// TwinCAT 3 PLC project SlaveController
// ProgramVersion: 3.1.4024.0
// libraries:
//   Tc2_EtherCAT, * (Beckhoff Automation GmbH)
//   Tc2_Math, * (Beckhoff Automation GmbH)
//   Tc2_Standard, * (Beckhoff Automation GmbH)
//   Tc2_System, * (Beckhoff Automation GmbH)
//   Tc2_Utilities, * (Beckhoff Automation GmbH)
//   Tc3_Module, * (Beckhoff Automation GmbH)
// project tree:
//   AgiMaths/Frames/ DHTrans.TcPOU (not stored), invFrame.TcPOU (not stored), rotX.TcPOU (not stored), rotY.TcPOU (not stored), rotZ.TcPOU (not stored), transform.TcPOU (not stored)
//   AgiMaths/MatrixLib/ angAxis2Rot.TcPOU (not stored), cross.TcPOU (not stored), Det5.TcPOU (not stored), Det6.TcPOU (not stored), Det7.TcPOU (not stored), invMat2.TcPOU (not stored), invMat6.TcPOU (not stored), invMat6Old.TcPOU (not stored), invMat3.TcPOU (not stored), invMat7.TcPOU (not stored), Mat3T.TcPOU (not stored), matAdd.TcPOU (not stored), matMultiNum.TcPOU (not stored), matMultiply.TcPOU (not stored), matMultiVec.TcPOU (not stored), matSelfAdd.TcPOU (not stored), vecDot.TcPOU (not stored), vecSelfAdd.TcPOU (not stored), matSelfSub.TcPOU (not stored), matSub.TcPOU (not stored), matTranspose.TcPOU (not stored), rot2AngAxis.TcPOU (not stored), vecAdd.TcPOU (not stored), norm.TcPOU (not stored), normalize.TcPOU (not stored), vecSelfMultiNum.TcPOU (not stored), vecMultiNum.TcPOU (not stored), vecSelfSub.TcPOU (not stored), vecSub.TcPOU (not stored)
//   AgiMaths/ sign.TcPOU (not stored), addVec7.TcPOU (not stored), atan2.TcPOU (not stored), cot.TcPOU (not stored)
//   DUTs/Enum/ E_ArmLightCtrlWord.TcDUT (not stored), E_CartJointState.TcDUT, E_EndoscopeType.TcDUT (not stored), E_EndoscopePosture.TcDUT (not stored), E_InstrumentType.TcDUT (not stored), E_MasterArmState.TcDUT (not stored), E_MatchedSlaveArmIdx.TcDUT (not stored), E_SetupArmState.TcDUT (not stored), E_SlaveArmState.TcDUT (not stored), E_DriverCtrlWord.TcDUT, E_DriverOPMode.TcDUT (not stored), E_DriverStatusWord.TcDUT (not stored)
//   DUTs/Structure/MasterSlaveCommunication/ ST_MasterStatus.TcDUT (not stored), ST_SlaveStatus.TcDUT (not stored)
//   DUTs/Structure/ ST_CartInputDataPool.TcDUT (not stored), ST_EtherCATState.TcDUT (not stored), ST_InstruOnChipData.TcDUT (not stored), ST_InstruStatus.TcDUT (not stored), ST_SetupArmCtrlCmds.TcDUT (not stored), ST_SetupInputDataPool.TcDUT (not stored), ST_SlaveArmCtrlCmds.TcDUT (not stored), ST_SlaveInputDataPool.TcDUT (not stored), ST_InstruKinematicParam.TcDUT (not stored), ST_Frame.TcDUT (not stored)
//   DUTs/Structure/TasksCommunication/ ST_CartJointData.TcDUT (not stored), ST_CartMotorInput.TcDUT (not stored), ST_CartMotorOutput.TcDUT (not stored), ST_CartStatus.TcDUT (not stored), ST_CartUIData.TcDUT (not stored), ST_SetupStatus.TcDUT (not stored), ST_SetupJointData.TcDUT (not stored), ST_SlaveDynaData.TcDUT (not stored), ST_SlaveUIData.TcDUT, ST_MasterJointData.TcDUT (not stored), ST_MotorInputs.TcDUT (not stored), ST_MotorOutputs.TcDUT (not stored), ST_SlaveJointData.TcDUT (not stored), ST_SafetyData.TcDUT (not stored)
//   DUTs/Structure/UICommunication/ ST_cartOperation.TcDUT (not stored), ST_instruInfomation.TcDUT (not stored), ST_robotStateMachine.TcDUT (not stored), ST_uiControl.TcDUT (not stored)
//   DUTs/Type/ Mat23.TcDUT (not stored), Mat2d.TcDUT (not stored), Mat32.TcDUT (not stored), Mat34.TcDUT (not stored), Mat53.TcDUT (not stored), Mat37.TcDUT (not stored), Mat43.TcDUT (not stored), Mat45.TcDUT (not stored), Mat35.TcDUT (not stored), Mat4d.TcDUT (not stored), Mat5d.TcDUT (not stored), Mat67.TcDUT (not stored), Mat6d.TcDUT (not stored), Mat76.TcDUT (not stored), Mat7d.TcDUT (not stored), Vec13d.TcDUT (not stored), Vec13di.TcDUT (not stored), Vec2d.TcDUT (not stored), Vec2i.TcDUT (not stored), Vec4b.TcDUT (not stored), Vec4d.TcDUT (not stored), Vec4i.TcDUT (not stored), Vec5b.TcDUT (not stored), Vec5d.TcDUT (not stored), Vec5i.TcDUT (not stored), Vec6b.TcDUT (not stored), Vec6i.TcDUT (not stored), Vec8b.TcDUT (not stored), Vec8d.TcDUT (not stored), Vec8di.TcDUT (not stored), Vec8i.TcDUT (not stored), Mat3d.TcDUT (not stored), Vec3d.TcDUT (not stored), Vec6d.TcDUT (not stored), Vec7d.TcDUT (not stored), Vec7i.TcDUT (not stored)
//   FBs_Auxiliary/ FB_cartJntDisenableDetect.TcPOU (not stored), FB_cartJntEnableDetect.TcPOU (not stored), FB_InstruNearDetect.TcPOU (not stored), FB_IOCheck.TcPOU (not stored), FB_IOToggleCheck.TcPOU (not stored), FB_rotaButtonDetect.TcPOU (not stored), FB_setupAdjustDetect.TcPOU (not stored), FB_setupJnt5AdjustDetect.TcPOU, FB_masterConnectionCheck.TcPOU (not stored), FB_TON.TcPOU (not stored), FB_trocarDetect.TcPOU (not stored), FB_PanelDetect.TcPOU, FB_InstrumentDetect.TcPOU, FB_AdjustDetect.TcPOU (not stored)
//   FBs_BasicControllers/ FB_dither.TcPOU (not stored), FB_BasicInstruControl.TcPOU (not stored), FBMacroJntControl.TcPOU (not stored), FB_UltrosonicKnifeControl.TcPOU (not stored), FB_PID.TcPOU (not stored)
//   FBs_CartControlles/ FB_CartCtrlAdjust.TcPOU, FB_CartCtrlAsepticDeploy.TcPOU (not stored), FB_CartCtrlBase.TcPOU (not stored), FB_CartCtrlError.TcPOU (not stored), FB_CartCtrlInit.TcPOU (not stored), FB_CartCtrlInSurgery.TcPOU (not stored), FB_CartCtrlMotionCar.TcPOU (not stored), FB_CartCtrlReady.TcPOU (not stored), FB_CartCtrlRotaOverhang.TcPOU (not stored), FB_CartCtrlSlowDown.TcPOU, FB_CartCtrlStandColuAdjust.TcPOU (not stored), FB_CartSupporLeg.TcPOU, I_CartJointCtrl.TcIO (not stored)
//   FBs_RobotDynamics/ FB_SlaveDynamic.TcPOU (not stored), FB_SlaveGravity.TcPOU (not stored), FB_SetupGravity.TcPOU
//   FBs_Robots/ FB_CartJoint.TcPOU, FB_CartRobot.TcPOU, FB_Instrument.TcPOU, FB_JointBase.TcPOU, FB_SetupArm.TcPOU, FB_SlaveCart.TcPOU, FB_SlaveJoint.TcPOU, FB_SetupJoint.TcPOU (not stored), FB_SetupRobot.TcPOU (not stored), FB_SlaveArm.TcPOU (not stored), FB_SlaveRobot.TcPOU
//   FBs_SetupControllers/ FB_SetupCtrlDisable.TcPOU (not stored), FB_SetupCtrlJnt5GraCali.TcPOU (not stored), FB_SetupCtrlHold.TcPOU (not stored), FB_SetupCtrlManualAdjust.TcPOU, FB_SetupCtrlPerformance.TcPOU (not stored), FB_SetupArmCtrlBase.TcPOU (not stored), FB_SetupCtrlAutoAdjust.TcPOU (not stored), FB_SetupCtrlCart.TcPOU (not stored), FB_SetupCtrlError.TcPOU (not stored), FB_SetupCtrlJnt3GraCali.TcPOU (not stored), FB_SetupCtrlInit.TcPOU (not stored), FB_SetupCtrlPackage.TcPOU (not stored), FB_SetupCtrlSelfCheck.TcPOU (not stored), I_SetupArmCtrl.TcIO (not stored)
//   FBs_SlaveControllers/ FB_SlaveCtrlDisable.TcPOU (not stored), FB_SlaveCtrlInstruInvasion.TcPOU (not stored), FB_SlaveCtrlInstruRetract.TcPOU (not stored), FB_SlaveCtrlInstruCali.TcPOU (not stored), FB_SlaveCtrlPerformance.TcPOU (not stored), FB_SlaveCtrlScopeToggle.TcPOU (not stored), FB_SlaveCtrlStop.TcPOU (not stored), FB_SlaveCtrlTest.TcPOU (not stored), FB_SlaveCtrlPackage.TcPOU (not stored), FB_SlaveCtrlEndoscope.TcPOU (not stored), FB_SlaveCtrlCart.TcPOU (not stored), FB_SlaveCtrlScopeReady.TcPOU (not stored), FB_SlaveCtrlSelfCheck.TcPOU, FB_SlaveCtrlError.TcPOU (not stored), FB_SlaveCtrlInstruReady.TcPOU (not stored), FB_SlaveCtrlMasterSlave.TcPOU, FB_SlaveCtrlMountInstru.TcPOU, FB_SlaveCtrlAdjust.TcPOU (not stored), FB_SlaveCtrlMountPanel.TcPOU (not stored), FB_SlaveCtrlPanelReady.TcPOU (not stored), FB_SlaveCtrlGraCali.TcPOU (not stored), FB_SlaveCtrlInit.TcPOU (not stored), FB_SlaveCtrlStandBy.TcPOU (not stored), FB_SlaveArmCtrlBase.TcPOU (not stored), I_SlaveArmCtrl.TcIO (not stored)
//   FBs_TrajectoryPlanning/ FB_BasicDoubleS.TcPOU (not stored), FB_trajBase.TcPOU (not stored), FB_TrajMoveJ.TcPOU (not stored), FB_setupTrajMoveJ.TcPOU (not stored), linear_trajectory_with_quintic_polynomial_blends.TcPOU (not stored), quintic_spline_curve.TcPOU (not stored), Quintic_spline_curve_factor.TcPOU (not stored), TrapezoIDal_velocity_trajectory.TcPOU (not stored)
//   FBs_TrajectoryPlanning/OTG/ FB_secOrdTrajFilter.TcPOU (not stored), FB_thirdOrdTrajFilter.TcPOU (not stored)
//   FBs_Filters/ FB_LowPassFilter.TcPOU (not stored)
//   GVLs/CartJoints/ GVL_CartControlParameters.TcGVL, GVL_CartJointEncoderCaliData.TcGVL, GVL_CartMotorParameters.TcGVL
//   GVLs/configs/robot3/ GVL_CartJointEncoderCaliData_3.TcGVL (not stored), GVL_SetupArmDynamics_3.TcGVL (not stored), GVL_SlaveArmDynamics_3.TcGVL (not stored), GVL_SetupJointEncoderCaliData_3.TcGVL (not stored), GVL_SlaveJointEncoderCaliData_3.TcGVL (not stored)
//   GVLs/configs/robot5/ GVL_CartJointEncoderCaliData_5.TcGVL (not stored), GVL_SetupArmDynamics_5.TcGVL (not stored), GVL_SlaveArmDynamics_5.TcGVL (not stored), GVL_SetupJointEncoderCaliData_5.TcGVL (not stored), GVL_SlaveJointEncoderCaliData_5.TcGVL (not stored)
//   GVLs/configs/robot4/ GVL_SetupArmDynamics_4.TcGVL (not stored), GVL_SetupJointEncoderCaliData_4.TcGVL (not stored), GVL_SlaveArmDynamics_4.TcGVL (not stored), GVL_SlaveJointEncoderCaliData_4.TcGVL (not stored)
//   GVLs/configs/robot6/ GVL_CartJointEncoderCaliData_6.TcGVL (not stored), GVL_SetupArmDynamics_6.TcGVL (not stored), GVL_SetupJointEncoderCaliData_6.TcGVL (not stored), GVL_SlaveArmDynamics_6.TcGVL (not stored), GVL_SlaveJointEncoderCaliData_6.TcGVL (not stored)
//   GVLs/ GVL_InstruCtrlParams.TcGVL, GVL_interactUI.TcGVL, GVL_MathDefine.TcGVL (not stored), GVL_SafetyLogData.TcGVL, GVL_SafetyParameters.TcGVL, GVL_SystemParameters.TcGVL
//   GVLs/SetupArms/ GVL_SetupArmDynamics.TcGVL (not stored), GVL_SetupJointEncoderCaliData.TcGVL, GVL_SetupMotorParameters.TcGVL, GVL_SetupArmKinematic.TcGVL (not stored), GVL_SetupControlParameters.TcGVL (not stored)
//   GVLs/SlaveArms/ GVL_SlaveArmDynamics.TcGVL (not stored), GVL_SlaveArmKinematic.TcGVL (not stored), GVL_SlaveControlParameters.TcGVL, GVL_SlaveJointEncoderCaliData.TcGVL, GVL_SlaveMotorParameters.TcGVL
//   Mains/ CartControl.TcPOU, SafetyCheck.TcPOU, SetupArmControl.TcPOU (not stored), SlaveArmControl.TcPOU, RobotDynamics.TcPOU (not stored)
//   SafetyCheck/ ASSERT.TcPOU (not stored), Fb_dataRecord.TcPOU (not stored), FB_EtherCATCheck.TcPOU (not stored), Fb_SafetyCheck.TcPOU, FB_Writer.TcPOU (not stored)
//   SafetyCheck/ErrRecord/ checkDelay.TcDUT (not stored), checkDelayTime.TcDUT, checkInputVariable.TcDUT (not stored), checkPermit.TcDUT (not stored), ST_Buffer.TcDUT (not stored), T_Buffer.TcDUT (not stored)
//   Sandbox/ FB_SlaveCtrlMasterSlave_bak1.TcPOU (not stored), FB_SlaveCtrlMasterSlave_bak2.TcPOU (not stored)
//   / TaskCartControl.TcTTO (not stored), TaskDynamic.TcTTO (not stored), TaskSafetyCheck.TcTTO (not stored), TaskSetupArmControl.TcTTO (not stored), TaskSlaveArmControl.TcTTO (not stored)
// real-time tasks:
//   TASK TaskSlaveArmControl: cycle T#250us, priority 1, ADS port 350
//   TASK TaskDynamic: cycle T#1ms, priority 2, ADS port 351
//   TASK TaskSetupArmControl: cycle T#1ms, priority 3, ADS port 352
//   TASK TaskSafetyCheck: cycle T#1ms, priority 6, ADS port 353
//   TASK TaskCartControl: cycle T#1ms, priority 4, ADS port 354
// I/O:
//   DEVICE CU2508
//   DEVICE Cart, AmsNetId 169.254.45.61.8.1
//     CartJoint5 [MDDLN55BE]
//     CartJoint3 [MDDLN55BE]
//     CartJoint4 [MDDLN55BE]
//     CartJoint1 [AX58200_MotorControl_for_1axis]
//     CartJoint2 [AX58200_MotorControl_for_1axis]
//     RS232 [AX58200_CANFD]
//     CartJoint6 [AX58200_MotorControl_for_1axis]
//     CartJoint7 [AX58200_MotorControl_for_1axis]
//     CartJoint8 [AX58200_MotorControl_for_1axis]
//   DEVICE MSCommunication, AmsNetId 169.254.186.39.3.1
//     Term 20 (EK1100) [EK1100 EtherCAT Coupler (2A E-Bus)]
//       Term 21 (EL6695) [EL6695 EtherCAT Bridge terminal (Primary)]
//       Term 8 (EL9011) [EL9011 End Terminal]
//     Term 22 (EK1100) [EK1100 EtherCAT Coupler (2A E-Bus)]
//       Term 23 (EL6070) [EL6070 1Ch. Licensing-Terminal]
//       Term 24 (EL1008) [EL1008 8Ch. Dig. Input 24V, 3ms]
//       Term 25 (EL2008) [EL2008 8Ch. Dig. Output 24V, 0.5A]
//       Term 26 (EL3004) [EL3004 4Ch. Ana. Input +/-10V] (disabled)
//       Term 9 (EL9011) [EL9011 End Terminal]
//   DEVICE SlaveArm1, AmsNetId 169.254.223.120.10.1
//     Box 25 (CU2508) [CU2508 Ethernet Port]
//     SetupJoint12 [AX58200_MotorControl_for_1axis]
//     SetupJoint3 [AX58200_MotorControl_for_1axis]
//     SetupJoint45 [AX58200_MotorControl_Slave45]
//     SlaveJoint1 [AX58200_MotorControl_for_1axis]
//     SlaveJoint2 [AX58200_MotorControl_for_1axis]
//     SlaveJoint3 [AX58200_MotorControl_for_1axis]
//     SlaveJoint45 [AX58200_MotorControl_3axis]
//     SlaveJoint678 [AX58200_MotorControl_3axis]
//   DEVICE SlaveArm2, AmsNetId 192.168.2.91.4.1
//     Box 25 (CU2508) [CU2508 Ethernet Port]
//     SetupJoint12 [AX58200_MotorControl_for_1axis]
//     SetupJoint3 [AX58200_MotorControl_for_1axis]
//     SetupJoint45 [AX58200_MotorControl_Slave45]
//     SlaveJoint1 [AX58200_MotorControl_for_1axis]
//     SlaveJoint2 [AX58200_MotorControl_for_1axis]
//     SlaveJoint3 [AX58200_MotorControl_for_1axis]
//     SlaveJoint45 [AX58200_MotorControl_3axis]
//     SlaveJoint678 [AX58200_MotorControl_3axis]
//   DEVICE SlaveArm3, AmsNetId 192.168.2.91.6.1
//     Box 17 (CU2508) [CU2508 Ethernet Port]
//     SetupJoint12 [AX58200_MotorControl_for_1axis]
//     SetupJoint3 [AX58200_MotorControl_for_1axis]
//     SetupJoint45 [AX58200_MotorControl_Slave45]
//     SlaveJoint1 [AX58200_MotorControl_for_1axis]
//     SlaveJoint2 [AX58200_MotorControl_for_1axis]
//     SlaveJoint3 [AX58200_MotorControl_for_1axis]
//     SlaveJoint45 [AX58200_MotorControl_3axis]
//     SlaveJoint678 [AX58200_MotorControl_3axis]
//   DEVICE SlaveArm4, AmsNetId 192.168.2.91.5.1
//     Box 9 (CU2508) [CU2508 Ethernet Port]
//     SetupJoint12 [AX58200_MotorControl_for_1axis]
//     SetupJoint3 [AX58200_MotorControl_for_1axis]
//     SetupJoint45 [AX58200_MotorControl_Slave45]
//     SlaveJoint1 [AX58200_MotorControl_for_1axis]
//     SlaveJoint2 [AX58200_MotorControl_for_1axis]
//     SlaveJoint3 [AX58200_MotorControl_for_1axis]
//     SlaveJoint45 [AX58200_MotorControl_3axis]
//     SlaveJoint678 [AX58200_MotorControl_3axis]
// variable links:
//   SlaveController/SlaveController Instance <-> Cart/CartJoint1
//     TaskCartControl Inputs/CartControl.m_cartRobot.m_slaveCart.m_cartJoints[1].m_motorInputs/m_current <-> TxPdoMappingCspCsv/Torque actual value
//     TaskCartControl Inputs/CartControl.m_cartRobot.m_slaveCart.m_cartJoints[1].m_motorInputs/m_motorEncoder <-> TxPdoMappingCspCsv/Position actual value
//     TaskCartControl Inputs/CartControl.m_cartRobot.m_slaveCart.m_cartJoints[1].m_motorInputs/m_statusWord <-> TxPdoMappingCspCsv/Statusword
//     TaskCartControl Inputs/CartControl.m_cartRobot.m_slaveCart.m_cartJoints[5].m_motorInputs/m_linkEncoder <-> TxPdoMappingCspCsv/ENC2
//     TaskCartControl Outputs/CartControl.m_cartRobot.m_slaveCart.m_cartJoints[1].m_motorOutputs/m_cmdCurrent <-> RxPdoMappingCspCsv/Target torque
//     TaskCartControl Outputs/CartControl.m_cartRobot.m_slaveCart.m_cartJoints[1].m_motorOutputs/m_cmdMotorEncoder <-> RxPdoMappingCspCsv/Target position
//     TaskCartControl Outputs/CartControl.m_cartRobot.m_slaveCart.m_cartJoints[1].m_motorOutputs/m_controlWord <-> RxPdoMappingCspCsv/Controlword
//     TaskCartControl Outputs/CartControl.m_cartRobot.m_slaveCart.m_cartJoints[1].m_motorOutputs/m_opMode <-> RxPdoMappingCspCsv/Modes of operation
//   SlaveController/SlaveController Instance <-> Cart/CartJoint2
//     TaskCartControl Inputs/CartControl.m_cartRobot.m_slaveCart.m_cartJoints[2].m_motorInputs/m_current <-> TxPdoMappingCspCsv/Torque actual value
//     TaskCartControl Inputs/CartControl.m_cartRobot.m_slaveCart.m_cartJoints[2].m_motorInputs/m_motorEncoder <-> TxPdoMappingCspCsv/Position actual value
//     TaskCartControl Inputs/CartControl.m_cartRobot.m_slaveCart.m_cartJoints[2].m_motorInputs/m_statusWord <-> TxPdoMappingCspCsv/Statusword
//     TaskCartControl Outputs/CartControl.m_cartRobot.m_slaveCart.m_cartJoints[2].m_motorOutputs/m_cmdCurrent <-> RxPdoMappingCspCsv/Target torque
//     TaskCartControl Outputs/CartControl.m_cartRobot.m_slaveCart.m_cartJoints[2].m_motorOutputs/m_cmdMotorEncoder <-> RxPdoMappingCspCsv/Target position
//     TaskCartControl Outputs/CartControl.m_cartRobot.m_slaveCart.m_cartJoints[2].m_motorOutputs/m_controlWord <-> RxPdoMappingCspCsv/Controlword
//     TaskCartControl Outputs/CartControl.m_cartRobot.m_slaveCart.m_cartJoints[2].m_motorOutputs/m_opMode <-> RxPdoMappingCspCsv/Modes of operation
//   SlaveController/SlaveController Instance <-> Cart/CartJoint3
//     TaskCartControl Inputs/CartControl.m_cartRobot.m_slaveCart.m_cartJoints[3].m_cartMotorVelSongxia <-> Transmit PDO mapping 2/Velocity actual value
//     TaskCartControl Inputs/CartControl.m_cartRobot.m_slaveCart.m_cartJoints[3].m_motorInputs/m_statusWord <-> Transmit PDO mapping 2/Statusword
//     TaskCartControl Outputs/CartControl.m_cartRobot.m_slaveCart.m_cartJoints[3].m_cartMotorOutput/m_cmdVelMax <-> Receive PDO mapping 2/Max motor speed
//     TaskCartControl Outputs/CartControl.m_cartRobot.m_slaveCart.m_cartJoints[3].m_cartMotorOutput/m_cmdVelMzVelMode <-> Receive PDO mapping 2/Target velocity
//     TaskCartControl Outputs/CartControl.m_cartRobot.m_slaveCart.m_cartJoints[3].m_motorOutputs/m_controlWord <-> Receive PDO mapping 2/Controlword
//     TaskCartControl Outputs/CartControl.m_cartRobot.m_slaveCart.m_cartJoints[3].m_motorOutputs/m_opMode <-> Receive PDO mapping 2/Modes of operation
//   SlaveController/SlaveController Instance <-> Cart/CartJoint4
//     TaskCartControl Inputs/CartControl.m_cartRobot.m_slaveCart.m_cartJoints[4].m_cartMotorVelSongxia <-> Transmit PDO mapping 2/Velocity actual value
//     TaskCartControl Inputs/CartControl.m_cartRobot.m_slaveCart.m_cartJoints[4].m_motorInputs/m_statusWord <-> Transmit PDO mapping 2/Statusword
//     TaskCartControl Outputs/CartControl.m_cartRobot.m_slaveCart.m_cartJoints[4].m_cartMotorOutput/m_cmdVelMax <-> Receive PDO mapping 2/Max motor speed
//     TaskCartControl Outputs/CartControl.m_cartRobot.m_slaveCart.m_cartJoints[4].m_cartMotorOutput/m_cmdVelMzVelMode <-> Receive PDO mapping 2/Target velocity
//     TaskCartControl Outputs/CartControl.m_cartRobot.m_slaveCart.m_cartJoints[4].m_motorOutputs/m_controlWord <-> Receive PDO mapping 2/Controlword
//     TaskCartControl Outputs/CartControl.m_cartRobot.m_slaveCart.m_cartJoints[4].m_motorOutputs/m_opMode <-> Receive PDO mapping 2/Modes of operation
//   SlaveController/SlaveController Instance <-> Cart/CartJoint5
//     TaskCartControl Inputs/CartControl.m_cartRobot.m_slaveCart.m_cartJoints[5].m_motorInputs/m_motorEncoder <-> Transmit PDO mapping 1/Position actual value
//     TaskCartControl Inputs/CartControl.m_cartRobot.m_slaveCart.m_cartJoints[5].m_motorInputs/m_statusWord <-> Transmit PDO mapping 1/Statusword
//     TaskCartControl Outputs/CartControl.m_cartRobot.m_slaveCart.m_cartJoints[5].m_motorOutputs/m_cmdMotorEncoder <-> Receive PDO mapping 1/Target position
//     TaskCartControl Outputs/CartControl.m_cartRobot.m_slaveCart.m_cartJoints[5].m_motorOutputs/m_controlWord <-> Receive PDO mapping 1/Controlword
//     TaskCartControl Outputs/CartControl.m_cartRobot.m_slaveCart.m_cartJoints[5].m_motorOutputs/m_opMode <-> Receive PDO mapping 1/Modes of operation
//   SlaveController/SlaveController Instance <-> Cart/CartJoint6
//     TaskCartControl Inputs/CartControl.m_cartRobot.m_slaveCart.m_cartJoints[6].m_motorInputs/m_current <-> TxPdoMappingCspCsv/Torque actual value
//     TaskCartControl Inputs/CartControl.m_cartRobot.m_slaveCart.m_cartJoints[6].m_motorInputs/m_linkEncoder <-> TxPdoMappingCspCsv/ENC2
//     TaskCartControl Inputs/CartControl.m_cartRobot.m_slaveCart.m_cartJoints[6].m_motorInputs/m_motorEncoder <-> TxPdoMappingCspCsv/Position actual value
//     TaskCartControl Inputs/CartControl.m_cartRobot.m_slaveCart.m_cartJoints[6].m_motorInputs/m_statusWord <-> TxPdoMappingCspCsv/Statusword
//     TaskCartControl Outputs/CartControl.m_cartRobot.m_openHorizonLaser <-> RxPdoMappingCspCsv/Target velocity
//     TaskCartControl Outputs/CartControl.m_cartRobot.m_slaveCart.m_cartJoints[6].m_motorOutputs/m_cmdCurrent <-> RxPdoMappingCspCsv/Target torque
//     TaskCartControl Outputs/CartControl.m_cartRobot.m_slaveCart.m_cartJoints[6].m_motorOutputs/m_cmdMotorEncoder <-> RxPdoMappingCspCsv/Target position
//     TaskCartControl Outputs/CartControl.m_cartRobot.m_slaveCart.m_cartJoints[6].m_motorOutputs/m_controlWord <-> RxPdoMappingCspCsv/Controlword
//     TaskCartControl Outputs/CartControl.m_cartRobot.m_slaveCart.m_cartJoints[6].m_motorOutputs/m_opMode <-> RxPdoMappingCspCsv/Modes of operation
//   SlaveController/SlaveController Instance <-> Cart/CartJoint7
//     TaskCartControl Inputs/CartControl.m_cartRobot.m_slaveCart.m_cartJoints[7].m_motorInputs/m_current <-> TxPdoMappingCspCsv/Torque actual value
//     TaskCartControl Inputs/CartControl.m_cartRobot.m_slaveCart.m_cartJoints[7].m_motorInputs/m_driverError <-> TxPdoMappingCspCsv/digital input
//     TaskCartControl Inputs/CartControl.m_cartRobot.m_slaveCart.m_cartJoints[7].m_motorInputs/m_linkEncoder <-> TxPdoMappingCspCsv/ENC2
//     TaskCartControl Inputs/CartControl.m_cartRobot.m_slaveCart.m_cartJoints[7].m_motorInputs/m_motorEncoder <-> TxPdoMappingCspCsv/Position actual value
//     TaskCartControl Inputs/CartControl.m_cartRobot.m_slaveCart.m_cartJoints[7].m_motorInputs/m_statusWord <-> TxPdoMappingCspCsv/Statusword
//     TaskCartControl Outputs/CartControl.m_cartRobot.m_slaveCart.m_cartJoints[7].m_motorOutputs/m_cmdCurrent <-> RxPdoMappingCspCsv/Target torque
//     TaskCartControl Outputs/CartControl.m_cartRobot.m_slaveCart.m_cartJoints[7].m_motorOutputs/m_cmdMotorEncoder <-> RxPdoMappingCspCsv/Target position
//     TaskCartControl Outputs/CartControl.m_cartRobot.m_slaveCart.m_cartJoints[7].m_motorOutputs/m_controlWord <-> RxPdoMappingCspCsv/Controlword
//     TaskCartControl Outputs/CartControl.m_cartRobot.m_slaveCart.m_cartJoints[7].m_motorOutputs/m_opMode <-> RxPdoMappingCspCsv/Modes of operation
//   SlaveController/SlaveController Instance <-> Cart/CartJoint8
//     TaskCartControl Inputs/CartControl.m_cartRobot.m_slaveCart.m_cartJoints[8].m_motorInputs/m_current <-> TxPdoMappingCspCsv/Torque actual value
//     TaskCartControl Inputs/CartControl.m_cartRobot.m_slaveCart.m_cartJoints[8].m_motorInputs/m_driverError <-> TxPdoMappingCspCsv/digital input
//     TaskCartControl Inputs/CartControl.m_cartRobot.m_slaveCart.m_cartJoints[8].m_motorInputs/m_linkEncoder <-> TxPdoMappingCspCsv/ENC2
//     TaskCartControl Inputs/CartControl.m_cartRobot.m_slaveCart.m_cartJoints[8].m_motorInputs/m_motorEncoder <-> TxPdoMappingCspCsv/Position actual value
//     TaskCartControl Inputs/CartControl.m_cartRobot.m_slaveCart.m_cartJoints[8].m_motorInputs/m_statusWord <-> TxPdoMappingCspCsv/Statusword
//     TaskCartControl Outputs/CartControl.m_cartRobot.m_openCrossLaser <-> RxPdoMappingCspCsv/Target velocity
//     TaskCartControl Outputs/CartControl.m_cartRobot.m_slaveCart.m_cartJoints[8].m_motorOutputs/m_cmdCurrent <-> RxPdoMappingCspCsv/Target torque
//     TaskCartControl Outputs/CartControl.m_cartRobot.m_slaveCart.m_cartJoints[8].m_motorOutputs/m_cmdMotorEncoder <-> RxPdoMappingCspCsv/Target position
//     TaskCartControl Outputs/CartControl.m_cartRobot.m_slaveCart.m_cartJoints[8].m_motorOutputs/m_controlWord <-> RxPdoMappingCspCsv/Controlword
//     TaskCartControl Outputs/CartControl.m_cartRobot.m_slaveCart.m_cartJoints[8].m_motorOutputs/m_opMode <-> RxPdoMappingCspCsv/Modes of operation
//   SlaveController/SlaveController Instance <-> Cart/RS232
//     TaskCartControl Inputs/CartControl.m_cartRobot.m_slaveCart.m_driveForce[1] <-> TxPdoMappingCspCsv/FX
//     TaskCartControl Inputs/CartControl.m_cartRobot.m_slaveCart.m_driveForce[2] <-> TxPdoMappingCspCsv/FY
//     TaskCartControl Inputs/CartControl.m_cartRobot.m_slaveCart.m_driveForce[3] <-> TxPdoMappingCspCsv/MZ
//     TaskCartControl Inputs/CartControl.m_cartRobot.m_slaveCart.m_joystickSignalIO[1] <-> TxPdoMappingCspCsv/D
//     TaskCartControl Inputs/CartControl.m_cartRobot.m_slaveCart.m_joystickSignalIO[2] <-> TxPdoMappingCspCsv/B
//     TaskCartControl Inputs/CartControl.m_cartRobot.m_slaveCart.m_joystickSignalIO[3] <-> TxPdoMappingCspCsv/A
//     TaskCartControl Inputs/CartControl.m_cartRobot.m_slaveCart.m_joystickSignalIO[4] <-> TxPdoMappingCspCsv/C
//   SlaveController/SlaveController Instance <-> MSCommunication/Term 20 (EK1100)/Term 21 (EL6695)
//     TaskSafetyCheck Inputs/SafetyCheck.m_masterRobotData <-> IO Inputs/MasterRobotData
//     TaskSlaveArmControl Inputs/SlaveArmControl.m_masterRobotData <-> IO Inputs/MasterRobotData
//     TaskSlaveArmControl Outputs/SlaveArmControl.m_slaveRobotData <-> IO Outputs/SlaveRobotData
//   SlaveController/SlaveController Instance <-> MSCommunication/Term 22 (EK1100)/Term 24 (EL1008)
//     TaskCartControl Inputs/CartControl.m_cartRobot.m_carHandChassisDriveUnlock[1] <-> Channel 5/Input
//     TaskCartControl Inputs/CartControl.m_cartRobot.m_carHandChassisDriveUnlock[2] <-> Channel 6/Input
//     TaskCartControl Inputs/CartControl.m_cartRobot.m_slaveCart.m_drivingLeverSensorAuto <-> Channel 8/Input
//     TaskCartControl Inputs/CartControl.m_cartRobot.m_slaveCart.m_drivingLeverSensorManual <-> Channel 7/Input
//     TaskCartControl Inputs/CartControl.m_cartRobot.m_slaveCart.m_stabilizFootSensorLeft <-> Channel 3/Input
//     TaskCartControl Inputs/CartControl.m_cartRobot.m_slaveCart.m_stabilizFootSensorRight <-> Channel 4/Input
//     TaskSafetyCheck Inputs/SafetyCheck.m_emergencyStopButton <-> Channel 2/Input
//     TaskSlaveArmControl Inputs/SafetyCheck.m_stopButton <-> Channel 1/Input
//   SlaveController/SlaveController Instance <-> MSCommunication/Term 22 (EK1100)/Term 25 (EL2008)
//     TaskCartControl Outputs/CartControl.m_cartRobot.m_slaveCart.m_screwBreak <-> Channel 5/Output
//     TaskSafetyCheck Outputs/SafetyCheck.m_warningTone[{1..4}] <-> Channel {1..4}/Output  (4 links)
//   SlaveController/SlaveController Instance <-> SlaveArm1/SetupJoint12
//     TaskSetupArmControl Inputs/SetupArmControl.m_setupRobot.m_setupArms[1].m_joints[1].m_motorInputs/m_linkEncoder <-> TxPdoMappingCspCsv/ENC2
//     TaskSetupArmControl Inputs/SetupArmControl.m_setupRobot.m_setupArms[1].m_joints[1].m_motorInputs/m_statusWord <-> TxPdoMappingCspCsv/Statusword
//     TaskSetupArmControl Inputs/SetupArmControl.m_setupRobot.m_setupArms[1].m_joints[2].m_motorInputs/m_statusWord <-> TxPdoMappingCspCsv/Statusword
//     TaskSetupArmControl Inputs/SetupArmControl.m_setupRobot.m_setupArms[1].m_joints[2].m_motorInputs/m_linkEncoder <-> TxPdoMappingCspCsv/Velocity actual value
//     TaskSetupArmControl Outputs/SetupArmControl.m_setupRobot.m_setupArms[1].m_joints[1].m_motorOutputs/m_controlWord <-> RxPdoMappingCspCsv/Controlword
//     TaskSetupArmControl Outputs/SetupArmControl.m_setupRobot.m_setupArms[1].m_joints[1].m_motorOutputs/m_opMode <-> RxPdoMappingCspCsv/Modes of operation
//   SlaveController/SlaveController Instance <-> SlaveArm1/SetupJoint3
//     TaskSetupArmControl Inputs/SetupArmControl.m_setupRobot.m_setupArms[1].m_joints[3].m_motorInputs/m_current <-> TxPdoMappingCspCsv/Torque actual value
//     TaskSetupArmControl Inputs/SetupArmControl.m_setupRobot.m_setupArms[1].m_joints[3].m_motorInputs/m_linkEncoder <-> TxPdoMappingCspCsv/ENC2
//     TaskSetupArmControl Inputs/SetupArmControl.m_setupRobot.m_setupArms[1].m_joints[3].m_motorInputs/m_motorEncoder <-> TxPdoMappingCspCsv/Position actual value
//     TaskSetupArmControl Inputs/SetupArmControl.m_setupRobot.m_setupArms[1].m_joints[3].m_motorInputs/m_statusWord <-> TxPdoMappingCspCsv/Statusword
//     TaskSetupArmControl Outputs/SetupArmControl.m_setupRobot.m_setupArms[1].m_joints[3].m_motorOutputs/m_cmdCurrent <-> RxPdoMappingCspCsv/Target torque
//     TaskSetupArmControl Outputs/SetupArmControl.m_setupRobot.m_setupArms[1].m_joints[3].m_motorOutputs/m_cmdMotorEncoder <-> RxPdoMappingCspCsv/Target position
//     TaskSetupArmControl Outputs/SetupArmControl.m_setupRobot.m_setupArms[1].m_joints[3].m_motorOutputs/m_controlWord <-> RxPdoMappingCspCsv/Controlword
//     TaskSetupArmControl Outputs/SetupArmControl.m_setupRobot.m_setupArms[1].m_joints[3].m_motorOutputs/m_opMode <-> RxPdoMappingCspCsv/Modes of operation
//   SlaveController/SlaveController Instance <-> SlaveArm1/SetupJoint45
//     TaskSetupArmControl Inputs/SetupArmControl.m_setupRobot.m_setupArms[1].m_joints[4].m_motorInputs/m_current <-> TxPdoMappingCspCsv/Torque actual value
//     TaskSetupArmControl Inputs/SetupArmControl.m_setupRobot.m_setupArms[1].m_joints[4].m_motorInputs/m_linkEncoder <-> TxPdoMappingCspCsv/ENC2
//     TaskSetupArmControl Inputs/SetupArmControl.m_setupRobot.m_setupArms[1].m_joints[4].m_motorInputs/m_motorEncoder <-> TxPdoMappingCspCsv/Position actual value
//     TaskSetupArmControl Inputs/SetupArmControl.m_setupRobot.m_setupArms[1].m_joints[4].m_motorInputs/m_statusWord <-> TxPdoMappingCspCsv/Statusword
//     TaskSetupArmControl Inputs/SetupArmControl.m_setupRobot.m_setupArms[1].m_joints[5].m_motorInputs/m_current <-> TxPdoMappingCspCsv/Torque actual value for aix2
//     TaskSetupArmControl Inputs/SetupArmControl.m_setupRobot.m_setupArms[1].m_joints[5].m_motorInputs/m_linkEncoder <-> TxPdoMappingCspCsv/ENC2 for aix2
//     TaskSetupArmControl Inputs/SetupArmControl.m_setupRobot.m_setupArms[1].m_joints[5].m_motorInputs/m_motorEncoder <-> TxPdoMappingCspCsv/Position actual value for aix2
//     TaskSetupArmControl Inputs/SetupArmControl.m_setupRobot.m_setupArms[1].m_joints[5].m_motorInputs/m_statusWord <-> TxPdoMappingCspCsv/Statusword for aix2
//     TaskSetupArmControl Outputs/SetupArmControl.m_setupRobot.m_setupArms[1].m_joints[4].m_motorOutputs/m_cmdCurrent <-> RxPdoMappingCspCsv/Target torque
//     TaskSetupArmControl Outputs/SetupArmControl.m_setupRobot.m_setupArms[1].m_joints[4].m_motorOutputs/m_cmdMotorEncoder <-> RxPdoMappingCspCsv/Target position
//     TaskSetupArmControl Outputs/SetupArmControl.m_setupRobot.m_setupArms[1].m_joints[4].m_motorOutputs/m_controlWord <-> RxPdoMappingCspCsv/Controlword
//     TaskSetupArmControl Outputs/SetupArmControl.m_setupRobot.m_setupArms[1].m_joints[4].m_motorOutputs/m_opMode <-> RxPdoMappingCspCsv/Modes of operation
//     TaskSetupArmControl Outputs/SetupArmControl.m_setupRobot.m_setupArms[1].m_joints[5].m_motorOutputs/m_cmdCurrent <-> RxPdoMappingCspCsv/Target Torque value for aix2
//     TaskSetupArmControl Outputs/SetupArmControl.m_setupRobot.m_setupArms[1].m_joints[5].m_motorOutputs/m_cmdMotorEncoder <-> RxPdoMappingCspCsv/Target position value for aix2
//     TaskSetupArmControl Outputs/SetupArmControl.m_setupRobot.m_setupArms[1].m_joints[5].m_motorOutputs/m_controlWord <-> RxPdoMappingCspCsv/ControlWord for aix2
//   SlaveController/SlaveController Instance <-> SlaveArm1/SlaveJoint1
//     TaskCartControl Inputs/CartControl.m_cartRobot.m_slaveCart.m_carRotaOverhangIO[1] <-> TxPdoMappingCspCsv/digital input
//     TaskSlaveArmControl Inputs/SlaveArmControl.m_slaveRobot.m_slaveArms[1].m_joints[1].m_motorInputs/m_current <-> TxPdoMappingCspCsv/Torque actual value
//     TaskSlaveArmControl Inputs/SlaveArmControl.m_slaveRobot.m_slaveArms[1].m_joints[1].m_motorInputs/m_driverError <-> TxPdoMappingCspCsv/digital input
//     TaskSlaveArmControl Inputs/SlaveArmControl.m_slaveRobot.m_slaveArms[1].m_joints[1].m_motorInputs/m_electriAngleDev <-> TxPdoMappingCspCsv/Velocity actual value
//     TaskSlaveArmControl Inputs/SlaveArmControl.m_slaveRobot.m_slaveArms[1].m_joints[1].m_motorInputs/m_linkEncoder <-> TxPdoMappingCspCsv/ENC2
//     TaskSlaveArmControl Inputs/SlaveArmControl.m_slaveRobot.m_slaveArms[1].m_joints[1].m_motorInputs/m_motorEncoder <-> TxPdoMappingCspCsv/Position actual value
//     TaskSlaveArmControl Inputs/SlaveArmControl.m_slaveRobot.m_slaveArms[1].m_joints[1].m_motorInputs/m_statusWord <-> TxPdoMappingCspCsv/Statusword
//     TaskSlaveArmControl Outputs/SlaveArmControl.m_slaveRobot.m_slaveArms[1].m_joints[1].m_motorOutputs/m_cmdCurrent <-> RxPdoMappingCspCsv/Target torque
//     TaskSlaveArmControl Outputs/SlaveArmControl.m_slaveRobot.m_slaveArms[1].m_joints[1].m_motorOutputs/m_cmdMotorEncoder <-> RxPdoMappingCspCsv/Target position
//     TaskSlaveArmControl Outputs/SlaveArmControl.m_slaveRobot.m_slaveArms[1].m_joints[1].m_motorOutputs/m_controlWord <-> RxPdoMappingCspCsv/Controlword
//     TaskSlaveArmControl Outputs/SlaveArmControl.m_slaveRobot.m_slaveArms[1].m_joints[1].m_motorOutputs/m_opMode <-> RxPdoMappingCspCsv/Modes of operation
//   SlaveController/SlaveController Instance <-> SlaveArm1/SlaveJoint2
//     TaskSetupArmControl Outputs/SetupArmControl.m_setupRobot.m_setupArms[1].m_lightIO <-> RxPdoMappingCspCsv/Target velocity
//     TaskSlaveArmControl Inputs/SlaveArmControl.m_slaveRobot.m_slaveArms[1].m_joints[2].m_motorInputs/m_current <-> TxPdoMappingCspCsv/Torque actual value
//     TaskSlaveArmControl Inputs/SlaveArmControl.m_slaveRobot.m_slaveArms[1].m_joints[2].m_motorInputs/m_driverError <-> TxPdoMappingCspCsv/digital input
//     TaskSlaveArmControl Inputs/SlaveArmControl.m_slaveRobot.m_slaveArms[1].m_joints[2].m_motorInputs/m_electriAngleDev <-> TxPdoMappingCspCsv/Velocity actual value
//     TaskSlaveArmControl Inputs/SlaveArmControl.m_slaveRobot.m_slaveArms[1].m_joints[2].m_motorInputs/m_linkEncoder <-> TxPdoMappingCspCsv/ENC2
//     TaskSlaveArmControl Inputs/SlaveArmControl.m_slaveRobot.m_slaveArms[1].m_joints[2].m_motorInputs/m_motorEncoder <-> TxPdoMappingCspCsv/Position actual value
//     TaskSlaveArmControl Inputs/SlaveArmControl.m_slaveRobot.m_slaveArms[1].m_joints[2].m_motorInputs/m_statusWord <-> TxPdoMappingCspCsv/Statusword
//     TaskSlaveArmControl Outputs/SlaveArmControl.m_slaveRobot.m_slaveArms[1].m_joints[2].m_motorOutputs/m_cmdCurrent <-> RxPdoMappingCspCsv/Target torque
//     TaskSlaveArmControl Outputs/SlaveArmControl.m_slaveRobot.m_slaveArms[1].m_joints[2].m_motorOutputs/m_cmdMotorEncoder <-> RxPdoMappingCspCsv/Target position
//     TaskSlaveArmControl Outputs/SlaveArmControl.m_slaveRobot.m_slaveArms[1].m_joints[2].m_motorOutputs/m_controlWord <-> RxPdoMappingCspCsv/Controlword
//     TaskSlaveArmControl Outputs/SlaveArmControl.m_slaveRobot.m_slaveArms[1].m_joints[2].m_motorOutputs/m_opMode <-> RxPdoMappingCspCsv/Modes of operation
//   SlaveController/SlaveController Instance <-> SlaveArm1/SlaveJoint3
//     TaskCartControl Inputs/CartControl.m_cartRobot.m_slaveCart.m_trocarIO[1] <-> TxPdoMappingCspCsv/digital input
//     TaskSetupArmControl Inputs/SetupArmControl.m_setupRobot.m_setupArms[1].m_adjustIO <-> TxPdoMappingCspCsv/digital input
//     TaskSlaveArmControl Inputs/SlaveArmControl.m_slaveRobot.m_slaveArms[1].m_adjustIO <-> TxPdoMappingCspCsv/digital input
//     TaskSlaveArmControl Inputs/SlaveArmControl.m_slaveRobot.m_slaveArms[1].m_joints[3].m_motorInputs/m_current <-> TxPdoMappingCspCsv/Torque actual value
//     TaskSlaveArmControl Inputs/SlaveArmControl.m_slaveRobot.m_slaveArms[1].m_joints[3].m_motorInputs/m_electriAngleDev <-> TxPdoMappingCspCsv/Velocity actual value
//     TaskSlaveArmControl Inputs/SlaveArmControl.m_slaveRobot.m_slaveArms[1].m_joints[3].m_motorInputs/m_linkEncoder <-> TxPdoMappingCspCsv/ENC2
//     TaskSlaveArmControl Inputs/SlaveArmControl.m_slaveRobot.m_slaveArms[1].m_joints[3].m_motorInputs/m_motorEncoder <-> TxPdoMappingCspCsv/Position actual value
//     TaskSlaveArmControl Inputs/SlaveArmControl.m_slaveRobot.m_slaveArms[1].m_joints[3].m_motorInputs/m_statusWord <-> TxPdoMappingCspCsv/Statusword
//     TaskSlaveArmControl Outputs/SlaveArmControl.m_slaveRobot.m_slaveArms[1].m_joints[3].m_motorOutputs/m_cmdCurrent <-> RxPdoMappingCspCsv/Target torque
//     TaskSlaveArmControl Outputs/SlaveArmControl.m_slaveRobot.m_slaveArms[1].m_joints[3].m_motorOutputs/m_cmdMotorEncoder <-> RxPdoMappingCspCsv/Target position
//     TaskSlaveArmControl Outputs/SlaveArmControl.m_slaveRobot.m_slaveArms[1].m_joints[3].m_motorOutputs/m_controlWord <-> RxPdoMappingCspCsv/Controlword
//     TaskSlaveArmControl Outputs/SlaveArmControl.m_slaveRobot.m_slaveArms[1].m_joints[3].m_motorOutputs/m_opMode <-> RxPdoMappingCspCsv/Modes of operation
//   SlaveController/SlaveController Instance <-> SlaveArm1/SlaveJoint45
//     TaskSlaveArmControl Inputs/SlaveArmControl.m_slaveRobot.m_slaveArms[1].m_joints[4].m_motorInputs/m_current <-> TxPdoMappingCspCsv/Velocity actual value for aix2
//     TaskSlaveArmControl Inputs/SlaveArmControl.m_slaveRobot.m_slaveArms[1].m_joints[4].m_motorInputs/m_linkEncoder <-> TxPdoMappingCspCsv/ENC2 for aix2
//     TaskSlaveArmControl Inputs/SlaveArmControl.m_slaveRobot.m_slaveArms[1].m_joints[5].m_motorInputs/m_linkEncoder <-> TxPdoMappingCspCsv/ENC2 for aix3
//     TaskSlaveArmControl Inputs/SlaveArmControl.m_slaveRobot.m_slaveArms[1].m_joints[4].m_motorInputs/m_motorEncoder <-> TxPdoMappingCspCsv/Position actual value for aix2
//     TaskSlaveArmControl Inputs/SlaveArmControl.m_slaveRobot.m_slaveArms[1].m_joints[5].m_motorInputs/m_motorEncoder <-> TxPdoMappingCspCsv/Position actual value for aix3
//     TaskSlaveArmControl Inputs/SlaveArmControl.m_slaveRobot.m_slaveArms[1].m_joints[4].m_motorInputs/m_statusWord <-> TxPdoMappingCspCsv/Statusword
//     TaskSlaveArmControl Inputs/SlaveArmControl.m_slaveRobot.m_slaveArms[1].m_joints[5].m_motorInputs/m_statusWord <-> TxPdoMappingCspCsv/Statusword
//     TaskSlaveArmControl Inputs/SlaveArmControl.m_slaveRobot.m_slaveArms[1].m_joints[5].m_motorInputs/m_current <-> TxPdoMappingCspCsv/Torque actual value for aix3
//     TaskSlaveArmControl Inputs/SlaveArmControl.m_slaveRobot.m_slaveArms[1].m_panelInstrumentOnIO <-> TxPdoMappingCspCsv/digital input
//     TaskSlaveArmControl Outputs/SlaveArmControl.m_slaveRobot.m_slaveArms[1].m_joints[4].m_motorOutputs/m_cmdCurrent <-> RxPdoMappingCspCsv/Target Torque value for aix2
//     TaskSlaveArmControl Outputs/SlaveArmControl.m_slaveRobot.m_slaveArms[1].m_joints[5].m_motorOutputs/m_cmdCurrent <-> RxPdoMappingCspCsv/Target Torque value for aix3
//     TaskSlaveArmControl Outputs/SlaveArmControl.m_slaveRobot.m_slaveArms[1].m_joints[4].m_motorOutputs/m_cmdMotorEncoder <-> RxPdoMappingCspCsv/Target position value for aix2
//     TaskSlaveArmControl Outputs/SlaveArmControl.m_slaveRobot.m_slaveArms[1].m_joints[5].m_motorOutputs/m_cmdMotorEncoder <-> RxPdoMappingCspCsv/Target position value for aix3
//     TaskSlaveArmControl Outputs/SlaveArmControl.m_slaveRobot.m_slaveArms[1].m_joints[4].m_motorOutputs/m_controlWord <-> RxPdoMappingCspCsv/Controlword
//     TaskSlaveArmControl Outputs/SlaveArmControl.m_slaveRobot.m_slaveArms[1].m_joints[4].m_motorOutputs/m_opMode <-> RxPdoMappingCspCsv/Modes of operation
//   SlaveController/SlaveController Instance <-> SlaveArm1/SlaveJoint678
//     TaskSlaveArmControl Inputs/SlaveArmControl.m_slaveRobot.m_slaveArms[1].m_joints[6].m_motorInputs/m_current <-> TxPdoMappingCspCsv/Velocity actual value for aix2
//     TaskSlaveArmControl Inputs/SlaveArmControl.m_slaveRobot.m_slaveArms[1].m_joints[6].m_motorInputs/m_linkEncoder <-> TxPdoMappingCspCsv/ENC2 for aix2
//     TaskSlaveArmControl Inputs/SlaveArmControl.m_slaveRobot.m_slaveArms[1].m_joints[7].m_motorInputs/m_linkEncoder <-> TxPdoMappingCspCsv/ENC2 for aix3
//     TaskSlaveArmControl Inputs/SlaveArmControl.m_slaveRobot.m_slaveArms[1].m_joints[8].m_motorInputs/m_linkEncoder <-> TxPdoMappingCspCsv/ENC2 for aix1
//     TaskSlaveArmControl Inputs/SlaveArmControl.m_slaveRobot.m_slaveArms[1].m_joints[6].m_motorInputs/m_motorEncoder <-> TxPdoMappingCspCsv/Position actual value for aix2
//     TaskSlaveArmControl Inputs/SlaveArmControl.m_slaveRobot.m_slaveArms[1].m_joints[7].m_motorInputs/m_motorEncoder <-> TxPdoMappingCspCsv/Position actual value for aix3
//     TaskSlaveArmControl Inputs/SlaveArmControl.m_slaveRobot.m_slaveArms[1].m_joints[6].m_motorInputs/m_statusWord <-> TxPdoMappingCspCsv/Statusword
//     TaskSlaveArmControl Inputs/SlaveArmControl.m_slaveRobot.m_slaveArms[1].m_joints[7].m_motorInputs/m_statusWord <-> TxPdoMappingCspCsv/Statusword
//     TaskSlaveArmControl Inputs/SlaveArmControl.m_slaveRobot.m_slaveArms[1].m_joints[8].m_motorInputs/m_statusWord <-> TxPdoMappingCspCsv/Statusword
//     TaskSlaveArmControl Inputs/SlaveArmControl.m_slaveRobot.m_slaveArms[1].m_joints[7].m_motorInputs/m_current <-> TxPdoMappingCspCsv/Torque actual value for aix3
//     TaskSlaveArmControl Inputs/SlaveArmControl.m_slaveRobot.m_slaveArms[1].m_joints[8].m_motorInputs/m_current <-> TxPdoMappingCspCsv/Torque actual value
//     TaskSlaveArmControl Inputs/SlaveArmControl.m_slaveRobot.m_slaveArms[1].m_joints[8].m_motorInputs/m_motorEncoder <-> TxPdoMappingCspCsv/Position actual value
//     TaskSlaveArmControl Outputs/SlaveArmControl.m_slaveRobot.m_slaveArms[1].m_joints[6].m_motorOutputs/m_cmdCurrent <-> RxPdoMappingCspCsv/Target Torque value for aix2
//     TaskSlaveArmControl Outputs/SlaveArmControl.m_slaveRobot.m_slaveArms[1].m_joints[7].m_motorOutputs/m_cmdCurrent <-> RxPdoMappingCspCsv/Target Torque value for aix3
//     TaskSlaveArmControl Outputs/SlaveArmControl.m_slaveRobot.m_slaveArms[1].m_joints[6].m_motorOutputs/m_cmdMotorEncoder <-> RxPdoMappingCspCsv/Target position value for aix2
//     TaskSlaveArmControl Outputs/SlaveArmControl.m_slaveRobot.m_slaveArms[1].m_joints[7].m_motorOutputs/m_cmdMotorEncoder <-> RxPdoMappingCspCsv/Target position value for aix3
//     TaskSlaveArmControl Outputs/SlaveArmControl.m_slaveRobot.m_slaveArms[1].m_joints[6].m_motorOutputs/m_controlWord <-> RxPdoMappingCspCsv/Controlword
//     TaskSlaveArmControl Outputs/SlaveArmControl.m_slaveRobot.m_slaveArms[1].m_joints[6].m_motorOutputs/m_opMode <-> RxPdoMappingCspCsv/Modes of operation
//     TaskSlaveArmControl Outputs/SlaveArmControl.m_slaveRobot.m_slaveArms[1].m_joints[8].m_motorOutputs/m_cmdCurrent <-> RxPdoMappingCspCsv/Target Torque value
//     TaskSlaveArmControl Outputs/SlaveArmControl.m_slaveRobot.m_slaveArms[1].m_joints[8].m_motorOutputs/m_cmdMotorEncoder <-> RxPdoMappingCspCsv/Target position
//   SlaveController/SlaveController Instance <-> SlaveArm2/SetupJoint12
//     TaskSetupArmControl Inputs/SetupArmControl.m_setupRobot.m_setupArms[2].m_joints[1].m_motorInputs/m_linkEncoder <-> TxPdoMappingCspCsv/ENC2
//     TaskSetupArmControl Inputs/SetupArmControl.m_setupRobot.m_setupArms[2].m_joints[1].m_motorInputs/m_statusWord <-> TxPdoMappingCspCsv/Statusword
//     TaskSetupArmControl Inputs/SetupArmControl.m_setupRobot.m_setupArms[2].m_joints[2].m_motorInputs/m_statusWord <-> TxPdoMappingCspCsv/Statusword
//     TaskSetupArmControl Inputs/SetupArmControl.m_setupRobot.m_setupArms[2].m_joints[2].m_motorInputs/m_linkEncoder <-> TxPdoMappingCspCsv/Velocity actual value
//     TaskSetupArmControl Outputs/SetupArmControl.m_setupRobot.m_setupArms[2].m_joints[1].m_motorOutputs/m_controlWord <-> RxPdoMappingCspCsv/Controlword
//     TaskSetupArmControl Outputs/SetupArmControl.m_setupRobot.m_setupArms[2].m_joints[1].m_motorOutputs/m_opMode <-> RxPdoMappingCspCsv/Modes of operation
//   SlaveController/SlaveController Instance <-> SlaveArm2/SetupJoint3
//     TaskSetupArmControl Inputs/SetupArmControl.m_setupRobot.m_setupArms[2].m_joints[3].m_motorInputs/m_current <-> TxPdoMappingCspCsv/Torque actual value
//     TaskSetupArmControl Inputs/SetupArmControl.m_setupRobot.m_setupArms[2].m_joints[3].m_motorInputs/m_driverError <-> TxPdoMappingCspCsv/digital input
//     TaskSetupArmControl Inputs/SetupArmControl.m_setupRobot.m_setupArms[2].m_joints[3].m_motorInputs/m_linkEncoder <-> TxPdoMappingCspCsv/ENC2
//     TaskSetupArmControl Inputs/SetupArmControl.m_setupRobot.m_setupArms[2].m_joints[3].m_motorInputs/m_motorEncoder <-> TxPdoMappingCspCsv/Position actual value
//     TaskSetupArmControl Inputs/SetupArmControl.m_setupRobot.m_setupArms[2].m_joints[3].m_motorInputs/m_statusWord <-> TxPdoMappingCspCsv/Statusword
//     TaskSetupArmControl Outputs/SetupArmControl.m_setupRobot.m_setupArms[2].m_joints[3].m_motorOutputs/m_cmdCurrent <-> RxPdoMappingCspCsv/Target torque
//     TaskSetupArmControl Outputs/SetupArmControl.m_setupRobot.m_setupArms[2].m_joints[3].m_motorOutputs/m_cmdMotorEncoder <-> RxPdoMappingCspCsv/Target position
//     TaskSetupArmControl Outputs/SetupArmControl.m_setupRobot.m_setupArms[2].m_joints[3].m_motorOutputs/m_controlWord <-> RxPdoMappingCspCsv/Controlword
//     TaskSetupArmControl Outputs/SetupArmControl.m_setupRobot.m_setupArms[2].m_joints[3].m_motorOutputs/m_opMode <-> RxPdoMappingCspCsv/Modes of operation
//   SlaveController/SlaveController Instance <-> SlaveArm2/SetupJoint45
//     TaskSetupArmControl Inputs/SetupArmControl.m_setupRobot.m_setupArms[2].m_joints[4].m_motorInputs/m_current <-> TxPdoMappingCspCsv/Torque actual value
//     TaskSetupArmControl Inputs/SetupArmControl.m_setupRobot.m_setupArms[2].m_joints[4].m_motorInputs/m_driverError <-> TxPdoMappingCspCsv/digital input
//     TaskSetupArmControl Inputs/SetupArmControl.m_setupRobot.m_setupArms[2].m_joints[4].m_motorInputs/m_linkEncoder <-> TxPdoMappingCspCsv/ENC2
//     TaskSetupArmControl Inputs/SetupArmControl.m_setupRobot.m_setupArms[2].m_joints[4].m_motorInputs/m_motorEncoder <-> TxPdoMappingCspCsv/Position actual value
//     TaskSetupArmControl Inputs/SetupArmControl.m_setupRobot.m_setupArms[2].m_joints[4].m_motorInputs/m_statusWord <-> TxPdoMappingCspCsv/Statusword
//     TaskSetupArmControl Inputs/SetupArmControl.m_setupRobot.m_setupArms[2].m_joints[5].m_motorInputs/m_current <-> TxPdoMappingCspCsv/Torque actual value for aix2
//     TaskSetupArmControl Inputs/SetupArmControl.m_setupRobot.m_setupArms[2].m_joints[5].m_motorInputs/m_linkEncoder <-> TxPdoMappingCspCsv/ENC2 for aix2
//     TaskSetupArmControl Inputs/SetupArmControl.m_setupRobot.m_setupArms[2].m_joints[5].m_motorInputs/m_motorEncoder <-> TxPdoMappingCspCsv/Position actual value for aix2
//     TaskSetupArmControl Inputs/SetupArmControl.m_setupRobot.m_setupArms[2].m_joints[5].m_motorInputs/m_statusWord <-> TxPdoMappingCspCsv/Statusword for aix2
//     TaskSetupArmControl Outputs/SetupArmControl.m_setupRobot.m_setupArms[2].m_joints[4].m_motorOutputs/m_cmdCurrent <-> RxPdoMappingCspCsv/Target torque
//     TaskSetupArmControl Outputs/SetupArmControl.m_setupRobot.m_setupArms[2].m_joints[4].m_motorOutputs/m_cmdMotorEncoder <-> RxPdoMappingCspCsv/Target position
//     TaskSetupArmControl Outputs/SetupArmControl.m_setupRobot.m_setupArms[2].m_joints[4].m_motorOutputs/m_controlWord <-> RxPdoMappingCspCsv/Controlword
//     TaskSetupArmControl Outputs/SetupArmControl.m_setupRobot.m_setupArms[2].m_joints[4].m_motorOutputs/m_opMode <-> RxPdoMappingCspCsv/Modes of operation
//     TaskSetupArmControl Outputs/SetupArmControl.m_setupRobot.m_setupArms[2].m_joints[5].m_motorOutputs/m_cmdCurrent <-> RxPdoMappingCspCsv/Target Torque value for aix2
//     TaskSetupArmControl Outputs/SetupArmControl.m_setupRobot.m_setupArms[2].m_joints[5].m_motorOutputs/m_cmdMotorEncoder <-> RxPdoMappingCspCsv/Target position value for aix2
//     TaskSetupArmControl Outputs/SetupArmControl.m_setupRobot.m_setupArms[2].m_joints[5].m_motorOutputs/m_controlWord <-> RxPdoMappingCspCsv/ControlWord for aix2
//   SlaveController/SlaveController Instance <-> SlaveArm2/SlaveJoint1
//     TaskCartControl Inputs/CartControl.m_cartRobot.m_slaveCart.m_carRotaOverhangIO[2] <-> TxPdoMappingCspCsv/digital input
//     TaskSlaveArmControl Inputs/SlaveArmControl.m_slaveRobot.m_slaveArms[2].m_joints[1].m_motorInputs/m_current <-> TxPdoMappingCspCsv/Torque actual value
//     TaskSlaveArmControl Inputs/SlaveArmControl.m_slaveRobot.m_slaveArms[2].m_joints[1].m_motorInputs/m_driverError <-> TxPdoMappingCspCsv/digital input
//     TaskSlaveArmControl Inputs/SlaveArmControl.m_slaveRobot.m_slaveArms[2].m_joints[1].m_motorInputs/m_electriAngleDev <-> TxPdoMappingCspCsv/Velocity actual value
//     TaskSlaveArmControl Inputs/SlaveArmControl.m_slaveRobot.m_slaveArms[2].m_joints[1].m_motorInputs/m_linkEncoder <-> TxPdoMappingCspCsv/ENC2
//     TaskSlaveArmControl Inputs/SlaveArmControl.m_slaveRobot.m_slaveArms[2].m_joints[1].m_motorInputs/m_motorEncoder <-> TxPdoMappingCspCsv/Position actual value
//     TaskSlaveArmControl Inputs/SlaveArmControl.m_slaveRobot.m_slaveArms[2].m_joints[1].m_motorInputs/m_statusWord <-> TxPdoMappingCspCsv/Statusword
//     TaskSlaveArmControl Outputs/SlaveArmControl.m_slaveRobot.m_slaveArms[2].m_joints[1].m_motorOutputs/m_cmdCurrent <-> RxPdoMappingCspCsv/Target torque
//     TaskSlaveArmControl Outputs/SlaveArmControl.m_slaveRobot.m_slaveArms[2].m_joints[1].m_motorOutputs/m_cmdMotorEncoder <-> RxPdoMappingCspCsv/Target position
//     TaskSlaveArmControl Outputs/SlaveArmControl.m_slaveRobot.m_slaveArms[2].m_joints[1].m_motorOutputs/m_controlWord <-> RxPdoMappingCspCsv/Controlword
//     TaskSlaveArmControl Outputs/SlaveArmControl.m_slaveRobot.m_slaveArms[2].m_joints[1].m_motorOutputs/m_opMode <-> RxPdoMappingCspCsv/Modes of operation
//   SlaveController/SlaveController Instance <-> SlaveArm2/SlaveJoint2
//     TaskSetupArmControl Outputs/SetupArmControl.m_setupRobot.m_setupArms[2].m_lightIO <-> RxPdoMappingCspCsv/Target velocity
//     TaskSlaveArmControl Inputs/SlaveArmControl.m_slaveRobot.m_slaveArms[2].m_joints[2].m_motorInputs/m_current <-> TxPdoMappingCspCsv/Torque actual value
//     TaskSlaveArmControl Inputs/SlaveArmControl.m_slaveRobot.m_slaveArms[2].m_joints[2].m_motorInputs/m_driverError <-> TxPdoMappingCspCsv/digital input
//     TaskSlaveArmControl Inputs/SlaveArmControl.m_slaveRobot.m_slaveArms[2].m_joints[2].m_motorInputs/m_electriAngleDev <-> TxPdoMappingCspCsv/Velocity actual value
//     TaskSlaveArmControl Inputs/SlaveArmControl.m_slaveRobot.m_slaveArms[2].m_joints[2].m_motorInputs/m_linkEncoder <-> TxPdoMappingCspCsv/ENC2
//     TaskSlaveArmControl Inputs/SlaveArmControl.m_slaveRobot.m_slaveArms[2].m_joints[2].m_motorInputs/m_motorEncoder <-> TxPdoMappingCspCsv/Position actual value
//     TaskSlaveArmControl Inputs/SlaveArmControl.m_slaveRobot.m_slaveArms[2].m_joints[2].m_motorInputs/m_statusWord <-> TxPdoMappingCspCsv/Statusword
//     TaskSlaveArmControl Outputs/SlaveArmControl.m_slaveRobot.m_slaveArms[2].m_joints[2].m_motorOutputs/m_cmdCurrent <-> RxPdoMappingCspCsv/Target torque
//     TaskSlaveArmControl Outputs/SlaveArmControl.m_slaveRobot.m_slaveArms[2].m_joints[2].m_motorOutputs/m_cmdMotorEncoder <-> RxPdoMappingCspCsv/Target position
//     TaskSlaveArmControl Outputs/SlaveArmControl.m_slaveRobot.m_slaveArms[2].m_joints[2].m_motorOutputs/m_controlWord <-> RxPdoMappingCspCsv/Controlword
//     TaskSlaveArmControl Outputs/SlaveArmControl.m_slaveRobot.m_slaveArms[2].m_joints[2].m_motorOutputs/m_opMode <-> RxPdoMappingCspCsv/Modes of operation
//   SlaveController/SlaveController Instance <-> SlaveArm2/SlaveJoint3
//     TaskCartControl Inputs/CartControl.m_cartRobot.m_slaveCart.m_trocarIO[2] <-> TxPdoMappingCspCsv/digital input
//     TaskSetupArmControl Inputs/SetupArmControl.m_setupRobot.m_setupArms[2].m_adjustIO <-> TxPdoMappingCspCsv/digital input
//     TaskSlaveArmControl Inputs/SlaveArmControl.m_slaveRobot.m_slaveArms[2].m_adjustIO <-> TxPdoMappingCspCsv/digital input
//     TaskSlaveArmControl Inputs/SlaveArmControl.m_slaveRobot.m_slaveArms[2].m_joints[3].m_motorInputs/m_current <-> TxPdoMappingCspCsv/Torque actual value
//     TaskSlaveArmControl Inputs/SlaveArmControl.m_slaveRobot.m_slaveArms[2].m_joints[3].m_motorInputs/m_linkEncoder <-> TxPdoMappingCspCsv/ENC2
//     TaskSlaveArmControl Inputs/SlaveArmControl.m_slaveRobot.m_slaveArms[2].m_joints[3].m_motorInputs/m_motorEncoder <-> TxPdoMappingCspCsv/Position actual value
//     TaskSlaveArmControl Inputs/SlaveArmControl.m_slaveRobot.m_slaveArms[2].m_joints[3].m_motorInputs/m_statusWord <-> TxPdoMappingCspCsv/Statusword
//     TaskSlaveArmControl Outputs/SlaveArmControl.m_slaveRobot.m_slaveArms[2].m_joints[3].m_motorOutputs/m_cmdCurrent <-> RxPdoMappingCspCsv/Target torque
//     TaskSlaveArmControl Outputs/SlaveArmControl.m_slaveRobot.m_slaveArms[2].m_joints[3].m_motorOutputs/m_cmdMotorEncoder <-> RxPdoMappingCspCsv/Target position
//     TaskSlaveArmControl Outputs/SlaveArmControl.m_slaveRobot.m_slaveArms[2].m_joints[3].m_motorOutputs/m_controlWord <-> RxPdoMappingCspCsv/Controlword
//     TaskSlaveArmControl Outputs/SlaveArmControl.m_slaveRobot.m_slaveArms[2].m_joints[3].m_motorOutputs/m_opMode <-> RxPdoMappingCspCsv/Modes of operation
//   SlaveController/SlaveController Instance <-> SlaveArm2/SlaveJoint45
//     TaskSlaveArmControl Inputs/SlaveArmControl.m_slaveRobot.m_slaveArms[2].m_joints[4].m_motorInputs/m_current <-> TxPdoMappingCspCsv/Velocity actual value for aix2
//     TaskSlaveArmControl Inputs/SlaveArmControl.m_slaveRobot.m_slaveArms[2].m_joints[4].m_motorInputs/m_linkEncoder <-> TxPdoMappingCspCsv/ENC2 for aix2
//     TaskSlaveArmControl Inputs/SlaveArmControl.m_slaveRobot.m_slaveArms[2].m_joints[5].m_motorInputs/m_linkEncoder <-> TxPdoMappingCspCsv/ENC2 for aix3
//     TaskSlaveArmControl Inputs/SlaveArmControl.m_slaveRobot.m_slaveArms[2].m_joints[4].m_motorInputs/m_motorEncoder <-> TxPdoMappingCspCsv/Position actual value for aix2
//     TaskSlaveArmControl Inputs/SlaveArmControl.m_slaveRobot.m_slaveArms[2].m_joints[5].m_motorInputs/m_motorEncoder <-> TxPdoMappingCspCsv/Position actual value for aix3
//     TaskSlaveArmControl Inputs/SlaveArmControl.m_slaveRobot.m_slaveArms[2].m_joints[4].m_motorInputs/m_statusWord <-> TxPdoMappingCspCsv/Statusword
//     TaskSlaveArmControl Inputs/SlaveArmControl.m_slaveRobot.m_slaveArms[2].m_joints[5].m_motorInputs/m_statusWord <-> TxPdoMappingCspCsv/Statusword
//     TaskSlaveArmControl Inputs/SlaveArmControl.m_slaveRobot.m_slaveArms[2].m_joints[5].m_motorInputs/m_current <-> TxPdoMappingCspCsv/Torque actual value for aix3
//     TaskSlaveArmControl Inputs/SlaveArmControl.m_slaveRobot.m_slaveArms[2].m_panelInstrumentOnIO <-> TxPdoMappingCspCsv/digital input
//     TaskSlaveArmControl Outputs/SlaveArmControl.m_slaveRobot.m_slaveArms[2].m_joints[4].m_motorOutputs/m_cmdCurrent <-> RxPdoMappingCspCsv/Target Torque value for aix2
//     TaskSlaveArmControl Outputs/SlaveArmControl.m_slaveRobot.m_slaveArms[2].m_joints[5].m_motorOutputs/m_cmdCurrent <-> RxPdoMappingCspCsv/Target Torque value for aix3
//     TaskSlaveArmControl Outputs/SlaveArmControl.m_slaveRobot.m_slaveArms[2].m_joints[4].m_motorOutputs/m_cmdMotorEncoder <-> RxPdoMappingCspCsv/Target position value for aix2
//     TaskSlaveArmControl Outputs/SlaveArmControl.m_slaveRobot.m_slaveArms[2].m_joints[5].m_motorOutputs/m_cmdMotorEncoder <-> RxPdoMappingCspCsv/Target position value for aix3
//     TaskSlaveArmControl Outputs/SlaveArmControl.m_slaveRobot.m_slaveArms[2].m_joints[4].m_motorOutputs/m_controlWord <-> RxPdoMappingCspCsv/Controlword
//     TaskSlaveArmControl Outputs/SlaveArmControl.m_slaveRobot.m_slaveArms[2].m_joints[4].m_motorOutputs/m_opMode <-> RxPdoMappingCspCsv/Modes of operation
//   SlaveController/SlaveController Instance <-> SlaveArm2/SlaveJoint678
//     TaskSlaveArmControl Inputs/SlaveArmControl.m_slaveRobot.m_slaveArms[2].m_joints[6].m_motorInputs/m_current <-> TxPdoMappingCspCsv/Velocity actual value for aix2
//     TaskSlaveArmControl Inputs/SlaveArmControl.m_slaveRobot.m_slaveArms[2].m_joints[6].m_motorInputs/m_linkEncoder <-> TxPdoMappingCspCsv/ENC2 for aix2
//     TaskSlaveArmControl Inputs/SlaveArmControl.m_slaveRobot.m_slaveArms[2].m_joints[7].m_motorInputs/m_linkEncoder <-> TxPdoMappingCspCsv/ENC2 for aix3
//     TaskSlaveArmControl Inputs/SlaveArmControl.m_slaveRobot.m_slaveArms[2].m_joints[8].m_motorInputs/m_linkEncoder <-> TxPdoMappingCspCsv/ENC2 for aix1
//     TaskSlaveArmControl Inputs/SlaveArmControl.m_slaveRobot.m_slaveArms[2].m_joints[6].m_motorInputs/m_motorEncoder <-> TxPdoMappingCspCsv/Position actual value for aix2
//     TaskSlaveArmControl Inputs/SlaveArmControl.m_slaveRobot.m_slaveArms[2].m_joints[7].m_motorInputs/m_motorEncoder <-> TxPdoMappingCspCsv/Position actual value for aix3
//     TaskSlaveArmControl Inputs/SlaveArmControl.m_slaveRobot.m_slaveArms[2].m_joints[6].m_motorInputs/m_statusWord <-> TxPdoMappingCspCsv/Statusword
//     TaskSlaveArmControl Inputs/SlaveArmControl.m_slaveRobot.m_slaveArms[2].m_joints[7].m_motorInputs/m_statusWord <-> TxPdoMappingCspCsv/Statusword
//     TaskSlaveArmControl Inputs/SlaveArmControl.m_slaveRobot.m_slaveArms[2].m_joints[8].m_motorInputs/m_statusWord <-> TxPdoMappingCspCsv/Statusword
//     TaskSlaveArmControl Inputs/SlaveArmControl.m_slaveRobot.m_slaveArms[2].m_joints[7].m_motorInputs/m_current <-> TxPdoMappingCspCsv/Torque actual value for aix3
//     TaskSlaveArmControl Inputs/SlaveArmControl.m_slaveRobot.m_slaveArms[2].m_joints[8].m_motorInputs/m_current <-> TxPdoMappingCspCsv/Torque actual value
//     TaskSlaveArmControl Inputs/SlaveArmControl.m_slaveRobot.m_slaveArms[2].m_joints[8].m_motorInputs/m_motorEncoder <-> TxPdoMappingCspCsv/Position actual value
//     TaskSlaveArmControl Outputs/SlaveArmControl.m_slaveRobot.m_slaveArms[2].m_joints[6].m_motorOutputs/m_cmdCurrent <-> RxPdoMappingCspCsv/Target Torque value for aix2
//     TaskSlaveArmControl Outputs/SlaveArmControl.m_slaveRobot.m_slaveArms[2].m_joints[7].m_motorOutputs/m_cmdCurrent <-> RxPdoMappingCspCsv/Target Torque value for aix3
//     TaskSlaveArmControl Outputs/SlaveArmControl.m_slaveRobot.m_slaveArms[2].m_joints[6].m_motorOutputs/m_cmdMotorEncoder <-> RxPdoMappingCspCsv/Target position value for aix2
//     TaskSlaveArmControl Outputs/SlaveArmControl.m_slaveRobot.m_slaveArms[2].m_joints[7].m_motorOutputs/m_cmdMotorEncoder <-> RxPdoMappingCspCsv/Target position value for aix3
//     TaskSlaveArmControl Outputs/SlaveArmControl.m_slaveRobot.m_slaveArms[2].m_joints[6].m_motorOutputs/m_controlWord <-> RxPdoMappingCspCsv/Controlword
//     TaskSlaveArmControl Outputs/SlaveArmControl.m_slaveRobot.m_slaveArms[2].m_joints[6].m_motorOutputs/m_opMode <-> RxPdoMappingCspCsv/Modes of operation
//     TaskSlaveArmControl Outputs/SlaveArmControl.m_slaveRobot.m_slaveArms[2].m_joints[8].m_motorOutputs/m_cmdCurrent <-> RxPdoMappingCspCsv/Target Torque value
//     TaskSlaveArmControl Outputs/SlaveArmControl.m_slaveRobot.m_slaveArms[2].m_joints[8].m_motorOutputs/m_cmdMotorEncoder <-> RxPdoMappingCspCsv/Target position
//   SlaveController/SlaveController Instance <-> SlaveArm3/SetupJoint12
//     TaskSetupArmControl Inputs/SetupArmControl.m_setupRobot.m_setupArms[3].m_joints[1].m_motorInputs/m_linkEncoder <-> TxPdoMappingCspCsv/ENC2
//     TaskSetupArmControl Inputs/SetupArmControl.m_setupRobot.m_setupArms[3].m_joints[1].m_motorInputs/m_statusWord <-> TxPdoMappingCspCsv/Statusword
//     TaskSetupArmControl Inputs/SetupArmControl.m_setupRobot.m_setupArms[3].m_joints[2].m_motorInputs/m_statusWord <-> TxPdoMappingCspCsv/Statusword
//     TaskSetupArmControl Inputs/SetupArmControl.m_setupRobot.m_setupArms[3].m_joints[2].m_motorInputs/m_linkEncoder <-> TxPdoMappingCspCsv/Velocity actual value
//     TaskSetupArmControl Outputs/SetupArmControl.m_setupRobot.m_setupArms[3].m_joints[1].m_motorOutputs/m_controlWord <-> RxPdoMappingCspCsv/Controlword
//     TaskSetupArmControl Outputs/SetupArmControl.m_setupRobot.m_setupArms[3].m_joints[1].m_motorOutputs/m_opMode <-> RxPdoMappingCspCsv/Modes of operation
//   SlaveController/SlaveController Instance <-> SlaveArm3/SetupJoint3
//     TaskSetupArmControl Inputs/SetupArmControl.m_setupRobot.m_setupArms[3].m_joints[3].m_motorInputs/m_current <-> TxPdoMappingCspCsv/Torque actual value
//     TaskSetupArmControl Inputs/SetupArmControl.m_setupRobot.m_setupArms[3].m_joints[3].m_motorInputs/m_driverError <-> TxPdoMappingCspCsv/digital input
//     TaskSetupArmControl Inputs/SetupArmControl.m_setupRobot.m_setupArms[3].m_joints[3].m_motorInputs/m_linkEncoder <-> TxPdoMappingCspCsv/ENC2
//     TaskSetupArmControl Inputs/SetupArmControl.m_setupRobot.m_setupArms[3].m_joints[3].m_motorInputs/m_motorEncoder <-> TxPdoMappingCspCsv/Position actual value
//     TaskSetupArmControl Inputs/SetupArmControl.m_setupRobot.m_setupArms[3].m_joints[3].m_motorInputs/m_statusWord <-> TxPdoMappingCspCsv/Statusword
//     TaskSetupArmControl Outputs/SetupArmControl.m_setupRobot.m_setupArms[3].m_joints[3].m_motorOutputs/m_cmdCurrent <-> RxPdoMappingCspCsv/Target torque
//     TaskSetupArmControl Outputs/SetupArmControl.m_setupRobot.m_setupArms[3].m_joints[3].m_motorOutputs/m_cmdMotorEncoder <-> RxPdoMappingCspCsv/Target position
//     TaskSetupArmControl Outputs/SetupArmControl.m_setupRobot.m_setupArms[3].m_joints[3].m_motorOutputs/m_controlWord <-> RxPdoMappingCspCsv/Controlword
//     TaskSetupArmControl Outputs/SetupArmControl.m_setupRobot.m_setupArms[3].m_joints[3].m_motorOutputs/m_opMode <-> RxPdoMappingCspCsv/Modes of operation
//   SlaveController/SlaveController Instance <-> SlaveArm3/SetupJoint45
//     TaskSetupArmControl Inputs/SetupArmControl.m_setupRobot.m_setupArms[3].m_joints[4].m_motorInputs/m_current <-> TxPdoMappingCspCsv/Torque actual value
//     TaskSetupArmControl Inputs/SetupArmControl.m_setupRobot.m_setupArms[3].m_joints[4].m_motorInputs/m_driverError <-> TxPdoMappingCspCsv/digital input
//     TaskSetupArmControl Inputs/SetupArmControl.m_setupRobot.m_setupArms[3].m_joints[4].m_motorInputs/m_linkEncoder <-> TxPdoMappingCspCsv/ENC2
//     TaskSetupArmControl Inputs/SetupArmControl.m_setupRobot.m_setupArms[3].m_joints[4].m_motorInputs/m_motorEncoder <-> TxPdoMappingCspCsv/Position actual value
//     TaskSetupArmControl Inputs/SetupArmControl.m_setupRobot.m_setupArms[3].m_joints[4].m_motorInputs/m_statusWord <-> TxPdoMappingCspCsv/Statusword
//     TaskSetupArmControl Inputs/SetupArmControl.m_setupRobot.m_setupArms[3].m_joints[5].m_motorInputs/m_current <-> TxPdoMappingCspCsv/Torque actual value for aix2
//     TaskSetupArmControl Inputs/SetupArmControl.m_setupRobot.m_setupArms[3].m_joints[5].m_motorInputs/m_linkEncoder <-> TxPdoMappingCspCsv/ENC2 for aix2
//     TaskSetupArmControl Inputs/SetupArmControl.m_setupRobot.m_setupArms[3].m_joints[5].m_motorInputs/m_motorEncoder <-> TxPdoMappingCspCsv/Position actual value for aix2
//     TaskSetupArmControl Inputs/SetupArmControl.m_setupRobot.m_setupArms[3].m_joints[5].m_motorInputs/m_statusWord <-> TxPdoMappingCspCsv/Statusword for aix2
//     TaskSetupArmControl Outputs/SetupArmControl.m_setupRobot.m_setupArms[3].m_joints[4].m_motorOutputs/m_cmdCurrent <-> RxPdoMappingCspCsv/Target torque
//     TaskSetupArmControl Outputs/SetupArmControl.m_setupRobot.m_setupArms[3].m_joints[4].m_motorOutputs/m_cmdMotorEncoder <-> RxPdoMappingCspCsv/Target position
//     TaskSetupArmControl Outputs/SetupArmControl.m_setupRobot.m_setupArms[3].m_joints[4].m_motorOutputs/m_controlWord <-> RxPdoMappingCspCsv/Controlword
//     TaskSetupArmControl Outputs/SetupArmControl.m_setupRobot.m_setupArms[3].m_joints[4].m_motorOutputs/m_opMode <-> RxPdoMappingCspCsv/Modes of operation
//     TaskSetupArmControl Outputs/SetupArmControl.m_setupRobot.m_setupArms[3].m_joints[5].m_motorOutputs/m_cmdCurrent <-> RxPdoMappingCspCsv/Target Torque value for aix2
//     TaskSetupArmControl Outputs/SetupArmControl.m_setupRobot.m_setupArms[3].m_joints[5].m_motorOutputs/m_cmdMotorEncoder <-> RxPdoMappingCspCsv/Target position value for aix2
//     TaskSetupArmControl Outputs/SetupArmControl.m_setupRobot.m_setupArms[3].m_joints[5].m_motorOutputs/m_controlWord <-> RxPdoMappingCspCsv/ControlWord for aix2
//   SlaveController/SlaveController Instance <-> SlaveArm3/SlaveJoint1
//     TaskCartControl Inputs/CartControl.m_cartRobot.m_slaveCart.m_carRotaOverhangIO[3] <-> TxPdoMappingCspCsv/digital input
//     TaskSlaveArmControl Inputs/SlaveArmControl.m_slaveRobot.m_slaveArms[3].m_joints[1].m_motorInputs/m_current <-> TxPdoMappingCspCsv/Torque actual value
//     TaskSlaveArmControl Inputs/SlaveArmControl.m_slaveRobot.m_slaveArms[3].m_joints[1].m_motorInputs/m_driverError <-> TxPdoMappingCspCsv/digital input
//     TaskSlaveArmControl Inputs/SlaveArmControl.m_slaveRobot.m_slaveArms[3].m_joints[1].m_motorInputs/m_electriAngleDev <-> TxPdoMappingCspCsv/Velocity actual value
//     TaskSlaveArmControl Inputs/SlaveArmControl.m_slaveRobot.m_slaveArms[3].m_joints[1].m_motorInputs/m_linkEncoder <-> TxPdoMappingCspCsv/ENC2
//     TaskSlaveArmControl Inputs/SlaveArmControl.m_slaveRobot.m_slaveArms[3].m_joints[1].m_motorInputs/m_motorEncoder <-> TxPdoMappingCspCsv/Position actual value
//     TaskSlaveArmControl Inputs/SlaveArmControl.m_slaveRobot.m_slaveArms[3].m_joints[1].m_motorInputs/m_statusWord <-> TxPdoMappingCspCsv/Statusword
//     TaskSlaveArmControl Outputs/SlaveArmControl.m_slaveRobot.m_slaveArms[3].m_joints[1].m_motorOutputs/m_cmdCurrent <-> RxPdoMappingCspCsv/Target torque
//     TaskSlaveArmControl Outputs/SlaveArmControl.m_slaveRobot.m_slaveArms[3].m_joints[1].m_motorOutputs/m_cmdMotorEncoder <-> RxPdoMappingCspCsv/Target position
//     TaskSlaveArmControl Outputs/SlaveArmControl.m_slaveRobot.m_slaveArms[3].m_joints[1].m_motorOutputs/m_controlWord <-> RxPdoMappingCspCsv/Controlword
//     TaskSlaveArmControl Outputs/SlaveArmControl.m_slaveRobot.m_slaveArms[3].m_joints[1].m_motorOutputs/m_opMode <-> RxPdoMappingCspCsv/Modes of operation
//   SlaveController/SlaveController Instance <-> SlaveArm3/SlaveJoint2
//     TaskSetupArmControl Outputs/SetupArmControl.m_setupRobot.m_setupArms[3].m_lightIO <-> RxPdoMappingCspCsv/Target velocity
//     TaskSlaveArmControl Inputs/SlaveArmControl.m_slaveRobot.m_slaveArms[3].m_joints[2].m_motorInputs/m_current <-> TxPdoMappingCspCsv/Torque actual value
//     TaskSlaveArmControl Inputs/SlaveArmControl.m_slaveRobot.m_slaveArms[3].m_joints[2].m_motorInputs/m_driverError <-> TxPdoMappingCspCsv/digital input
//     TaskSlaveArmControl Inputs/SlaveArmControl.m_slaveRobot.m_slaveArms[3].m_joints[2].m_motorInputs/m_electriAngleDev <-> TxPdoMappingCspCsv/Velocity actual value
//     TaskSlaveArmControl Inputs/SlaveArmControl.m_slaveRobot.m_slaveArms[3].m_joints[2].m_motorInputs/m_linkEncoder <-> TxPdoMappingCspCsv/ENC2
//     TaskSlaveArmControl Inputs/SlaveArmControl.m_slaveRobot.m_slaveArms[3].m_joints[2].m_motorInputs/m_motorEncoder <-> TxPdoMappingCspCsv/Position actual value
//     TaskSlaveArmControl Inputs/SlaveArmControl.m_slaveRobot.m_slaveArms[3].m_joints[2].m_motorInputs/m_statusWord <-> TxPdoMappingCspCsv/Statusword
//     TaskSlaveArmControl Outputs/SlaveArmControl.m_slaveRobot.m_slaveArms[3].m_joints[2].m_motorOutputs/m_cmdCurrent <-> RxPdoMappingCspCsv/Target torque
//     TaskSlaveArmControl Outputs/SlaveArmControl.m_slaveRobot.m_slaveArms[3].m_joints[2].m_motorOutputs/m_cmdMotorEncoder <-> RxPdoMappingCspCsv/Target position
//     TaskSlaveArmControl Outputs/SlaveArmControl.m_slaveRobot.m_slaveArms[3].m_joints[2].m_motorOutputs/m_controlWord <-> RxPdoMappingCspCsv/Controlword
//     TaskSlaveArmControl Outputs/SlaveArmControl.m_slaveRobot.m_slaveArms[3].m_joints[2].m_motorOutputs/m_opMode <-> RxPdoMappingCspCsv/Modes of operation
//   SlaveController/SlaveController Instance <-> SlaveArm3/SlaveJoint3
//     TaskCartControl Inputs/CartControl.m_cartRobot.m_slaveCart.m_trocarIO[3] <-> TxPdoMappingCspCsv/digital input
//     TaskSetupArmControl Inputs/SetupArmControl.m_setupRobot.m_setupArms[3].m_adjustIO <-> TxPdoMappingCspCsv/digital input
//     TaskSlaveArmControl Inputs/SlaveArmControl.m_slaveRobot.m_slaveArms[3].m_adjustIO <-> TxPdoMappingCspCsv/digital input
//     TaskSlaveArmControl Inputs/SlaveArmControl.m_slaveRobot.m_slaveArms[3].m_joints[3].m_motorInputs/m_current <-> TxPdoMappingCspCsv/Torque actual value
//     TaskSlaveArmControl Inputs/SlaveArmControl.m_slaveRobot.m_slaveArms[3].m_joints[3].m_motorInputs/m_linkEncoder <-> TxPdoMappingCspCsv/ENC2
//     TaskSlaveArmControl Inputs/SlaveArmControl.m_slaveRobot.m_slaveArms[3].m_joints[3].m_motorInputs/m_motorEncoder <-> TxPdoMappingCspCsv/Position actual value
//     TaskSlaveArmControl Inputs/SlaveArmControl.m_slaveRobot.m_slaveArms[3].m_joints[3].m_motorInputs/m_statusWord <-> TxPdoMappingCspCsv/Statusword
//     TaskSlaveArmControl Outputs/SlaveArmControl.m_slaveRobot.m_slaveArms[3].m_joints[3].m_motorOutputs/m_cmdCurrent <-> RxPdoMappingCspCsv/Target torque
//     TaskSlaveArmControl Outputs/SlaveArmControl.m_slaveRobot.m_slaveArms[3].m_joints[3].m_motorOutputs/m_cmdMotorEncoder <-> RxPdoMappingCspCsv/Target position
//     TaskSlaveArmControl Outputs/SlaveArmControl.m_slaveRobot.m_slaveArms[3].m_joints[3].m_motorOutputs/m_controlWord <-> RxPdoMappingCspCsv/Controlword
//     TaskSlaveArmControl Outputs/SlaveArmControl.m_slaveRobot.m_slaveArms[3].m_joints[3].m_motorOutputs/m_opMode <-> RxPdoMappingCspCsv/Modes of operation
//   SlaveController/SlaveController Instance <-> SlaveArm3/SlaveJoint45
//     TaskSlaveArmControl Inputs/SlaveArmControl.m_slaveRobot.m_slaveArms[3].m_joints[4].m_motorInputs/m_current <-> TxPdoMappingCspCsv/Velocity actual value for aix2
//     TaskSlaveArmControl Inputs/SlaveArmControl.m_slaveRobot.m_slaveArms[3].m_joints[4].m_motorInputs/m_linkEncoder <-> TxPdoMappingCspCsv/ENC2 for aix2
//     TaskSlaveArmControl Inputs/SlaveArmControl.m_slaveRobot.m_slaveArms[3].m_joints[5].m_motorInputs/m_linkEncoder <-> TxPdoMappingCspCsv/ENC2 for aix3
//     TaskSlaveArmControl Inputs/SlaveArmControl.m_slaveRobot.m_slaveArms[3].m_joints[4].m_motorInputs/m_motorEncoder <-> TxPdoMappingCspCsv/Position actual value for aix2
//     TaskSlaveArmControl Inputs/SlaveArmControl.m_slaveRobot.m_slaveArms[3].m_joints[5].m_motorInputs/m_motorEncoder <-> TxPdoMappingCspCsv/Position actual value for aix3
//     TaskSlaveArmControl Inputs/SlaveArmControl.m_slaveRobot.m_slaveArms[3].m_joints[4].m_motorInputs/m_statusWord <-> TxPdoMappingCspCsv/Statusword
//     TaskSlaveArmControl Inputs/SlaveArmControl.m_slaveRobot.m_slaveArms[3].m_joints[5].m_motorInputs/m_statusWord <-> TxPdoMappingCspCsv/Statusword
//     TaskSlaveArmControl Inputs/SlaveArmControl.m_slaveRobot.m_slaveArms[3].m_joints[5].m_motorInputs/m_current <-> TxPdoMappingCspCsv/Torque actual value for aix3
//     TaskSlaveArmControl Inputs/SlaveArmControl.m_slaveRobot.m_slaveArms[3].m_panelInstrumentOnIO <-> TxPdoMappingCspCsv/digital input
//     TaskSlaveArmControl Outputs/SlaveArmControl.m_slaveRobot.m_slaveArms[3].m_joints[4].m_motorOutputs/m_cmdCurrent <-> RxPdoMappingCspCsv/Target Torque value for aix2
//     TaskSlaveArmControl Outputs/SlaveArmControl.m_slaveRobot.m_slaveArms[3].m_joints[5].m_motorOutputs/m_cmdCurrent <-> RxPdoMappingCspCsv/Target Torque value for aix3
//     TaskSlaveArmControl Outputs/SlaveArmControl.m_slaveRobot.m_slaveArms[3].m_joints[4].m_motorOutputs/m_cmdMotorEncoder <-> RxPdoMappingCspCsv/Target position value for aix2
//     TaskSlaveArmControl Outputs/SlaveArmControl.m_slaveRobot.m_slaveArms[3].m_joints[5].m_motorOutputs/m_cmdMotorEncoder <-> RxPdoMappingCspCsv/Target position value for aix3
//     TaskSlaveArmControl Outputs/SlaveArmControl.m_slaveRobot.m_slaveArms[3].m_joints[4].m_motorOutputs/m_controlWord <-> RxPdoMappingCspCsv/Controlword
//     TaskSlaveArmControl Outputs/SlaveArmControl.m_slaveRobot.m_slaveArms[3].m_joints[4].m_motorOutputs/m_opMode <-> RxPdoMappingCspCsv/Modes of operation
//   SlaveController/SlaveController Instance <-> SlaveArm3/SlaveJoint678
//     TaskSlaveArmControl Inputs/SlaveArmControl.m_slaveRobot.m_slaveArms[3].m_joints[6].m_motorInputs/m_current <-> TxPdoMappingCspCsv/Velocity actual value for aix2
//     TaskSlaveArmControl Inputs/SlaveArmControl.m_slaveRobot.m_slaveArms[3].m_joints[6].m_motorInputs/m_linkEncoder <-> TxPdoMappingCspCsv/ENC2 for aix2
//     TaskSlaveArmControl Inputs/SlaveArmControl.m_slaveRobot.m_slaveArms[3].m_joints[7].m_motorInputs/m_linkEncoder <-> TxPdoMappingCspCsv/ENC2 for aix3
//     TaskSlaveArmControl Inputs/SlaveArmControl.m_slaveRobot.m_slaveArms[3].m_joints[8].m_motorInputs/m_linkEncoder <-> TxPdoMappingCspCsv/ENC2 for aix1
//     TaskSlaveArmControl Inputs/SlaveArmControl.m_slaveRobot.m_slaveArms[3].m_joints[6].m_motorInputs/m_motorEncoder <-> TxPdoMappingCspCsv/Position actual value for aix2
//     TaskSlaveArmControl Inputs/SlaveArmControl.m_slaveRobot.m_slaveArms[3].m_joints[7].m_motorInputs/m_motorEncoder <-> TxPdoMappingCspCsv/Position actual value for aix3
//     TaskSlaveArmControl Inputs/SlaveArmControl.m_slaveRobot.m_slaveArms[3].m_joints[6].m_motorInputs/m_statusWord <-> TxPdoMappingCspCsv/Statusword
//     TaskSlaveArmControl Inputs/SlaveArmControl.m_slaveRobot.m_slaveArms[3].m_joints[7].m_motorInputs/m_statusWord <-> TxPdoMappingCspCsv/Statusword
//     TaskSlaveArmControl Inputs/SlaveArmControl.m_slaveRobot.m_slaveArms[3].m_joints[8].m_motorInputs/m_statusWord <-> TxPdoMappingCspCsv/Statusword
//     TaskSlaveArmControl Inputs/SlaveArmControl.m_slaveRobot.m_slaveArms[3].m_joints[7].m_motorInputs/m_current <-> TxPdoMappingCspCsv/Torque actual value for aix3
//     TaskSlaveArmControl Inputs/SlaveArmControl.m_slaveRobot.m_slaveArms[3].m_joints[8].m_motorInputs/m_current <-> TxPdoMappingCspCsv/Torque actual value
//     TaskSlaveArmControl Inputs/SlaveArmControl.m_slaveRobot.m_slaveArms[3].m_joints[8].m_motorInputs/m_motorEncoder <-> TxPdoMappingCspCsv/Position actual value
//     TaskSlaveArmControl Outputs/SlaveArmControl.m_slaveRobot.m_slaveArms[3].m_joints[6].m_motorOutputs/m_cmdCurrent <-> RxPdoMappingCspCsv/Target Torque value for aix2
//     TaskSlaveArmControl Outputs/SlaveArmControl.m_slaveRobot.m_slaveArms[3].m_joints[7].m_motorOutputs/m_cmdCurrent <-> RxPdoMappingCspCsv/Target Torque value for aix3
//     TaskSlaveArmControl Outputs/SlaveArmControl.m_slaveRobot.m_slaveArms[3].m_joints[6].m_motorOutputs/m_cmdMotorEncoder <-> RxPdoMappingCspCsv/Target position value for aix2
//     TaskSlaveArmControl Outputs/SlaveArmControl.m_slaveRobot.m_slaveArms[3].m_joints[7].m_motorOutputs/m_cmdMotorEncoder <-> RxPdoMappingCspCsv/Target position value for aix3
//     TaskSlaveArmControl Outputs/SlaveArmControl.m_slaveRobot.m_slaveArms[3].m_joints[6].m_motorOutputs/m_controlWord <-> RxPdoMappingCspCsv/Controlword
//     TaskSlaveArmControl Outputs/SlaveArmControl.m_slaveRobot.m_slaveArms[3].m_joints[6].m_motorOutputs/m_opMode <-> RxPdoMappingCspCsv/Modes of operation
//     TaskSlaveArmControl Outputs/SlaveArmControl.m_slaveRobot.m_slaveArms[3].m_joints[8].m_motorOutputs/m_cmdCurrent <-> RxPdoMappingCspCsv/Target Torque value
//     TaskSlaveArmControl Outputs/SlaveArmControl.m_slaveRobot.m_slaveArms[3].m_joints[8].m_motorOutputs/m_cmdMotorEncoder <-> RxPdoMappingCspCsv/Target position
//   SlaveController/SlaveController Instance <-> SlaveArm4/SetupJoint12
//     TaskSetupArmControl Inputs/SetupArmControl.m_setupRobot.m_setupArms[4].m_joints[1].m_motorInputs/m_linkEncoder <-> TxPdoMappingCspCsv/ENC2
//     TaskSetupArmControl Inputs/SetupArmControl.m_setupRobot.m_setupArms[4].m_joints[1].m_motorInputs/m_statusWord <-> TxPdoMappingCspCsv/Statusword
//     TaskSetupArmControl Inputs/SetupArmControl.m_setupRobot.m_setupArms[4].m_joints[2].m_motorInputs/m_statusWord <-> TxPdoMappingCspCsv/Statusword
//     TaskSetupArmControl Inputs/SetupArmControl.m_setupRobot.m_setupArms[4].m_joints[2].m_motorInputs/m_linkEncoder <-> TxPdoMappingCspCsv/Velocity actual value
//     TaskSetupArmControl Outputs/SetupArmControl.m_setupRobot.m_setupArms[4].m_joints[1].m_motorOutputs/m_controlWord <-> RxPdoMappingCspCsv/Controlword
//     TaskSetupArmControl Outputs/SetupArmControl.m_setupRobot.m_setupArms[4].m_joints[1].m_motorOutputs/m_opMode <-> RxPdoMappingCspCsv/Modes of operation
//   SlaveController/SlaveController Instance <-> SlaveArm4/SetupJoint3
//     TaskSetupArmControl Inputs/SetupArmControl.m_setupRobot.m_setupArms[4].m_joints[3].m_motorInputs/m_current <-> TxPdoMappingCspCsv/Torque actual value
//     TaskSetupArmControl Inputs/SetupArmControl.m_setupRobot.m_setupArms[4].m_joints[3].m_motorInputs/m_driverError <-> TxPdoMappingCspCsv/digital input
//     TaskSetupArmControl Inputs/SetupArmControl.m_setupRobot.m_setupArms[4].m_joints[3].m_motorInputs/m_linkEncoder <-> TxPdoMappingCspCsv/ENC2
//     TaskSetupArmControl Inputs/SetupArmControl.m_setupRobot.m_setupArms[4].m_joints[3].m_motorInputs/m_motorEncoder <-> TxPdoMappingCspCsv/Position actual value
//     TaskSetupArmControl Inputs/SetupArmControl.m_setupRobot.m_setupArms[4].m_joints[3].m_motorInputs/m_statusWord <-> TxPdoMappingCspCsv/Statusword
//     TaskSetupArmControl Outputs/SetupArmControl.m_setupRobot.m_setupArms[4].m_joints[3].m_motorOutputs/m_cmdCurrent <-> RxPdoMappingCspCsv/Target torque
//     TaskSetupArmControl Outputs/SetupArmControl.m_setupRobot.m_setupArms[4].m_joints[3].m_motorOutputs/m_cmdMotorEncoder <-> RxPdoMappingCspCsv/Target position
//     TaskSetupArmControl Outputs/SetupArmControl.m_setupRobot.m_setupArms[4].m_joints[3].m_motorOutputs/m_controlWord <-> RxPdoMappingCspCsv/Controlword
//     TaskSetupArmControl Outputs/SetupArmControl.m_setupRobot.m_setupArms[4].m_joints[3].m_motorOutputs/m_opMode <-> RxPdoMappingCspCsv/Modes of operation
//   SlaveController/SlaveController Instance <-> SlaveArm4/SetupJoint45
//     TaskSetupArmControl Inputs/SetupArmControl.m_setupRobot.m_setupArms[4].m_joints[4].m_motorInputs/m_current <-> TxPdoMappingCspCsv/Torque actual value
//     TaskSetupArmControl Inputs/SetupArmControl.m_setupRobot.m_setupArms[4].m_joints[4].m_motorInputs/m_driverError <-> TxPdoMappingCspCsv/digital input
//     TaskSetupArmControl Inputs/SetupArmControl.m_setupRobot.m_setupArms[4].m_joints[4].m_motorInputs/m_linkEncoder <-> TxPdoMappingCspCsv/ENC2
//     TaskSetupArmControl Inputs/SetupArmControl.m_setupRobot.m_setupArms[4].m_joints[4].m_motorInputs/m_motorEncoder <-> TxPdoMappingCspCsv/Position actual value
//     TaskSetupArmControl Inputs/SetupArmControl.m_setupRobot.m_setupArms[4].m_joints[4].m_motorInputs/m_statusWord <-> TxPdoMappingCspCsv/Statusword
//     TaskSetupArmControl Inputs/SetupArmControl.m_setupRobot.m_setupArms[4].m_joints[5].m_motorInputs/m_current <-> TxPdoMappingCspCsv/Torque actual value for aix2
//     TaskSetupArmControl Inputs/SetupArmControl.m_setupRobot.m_setupArms[4].m_joints[5].m_motorInputs/m_linkEncoder <-> TxPdoMappingCspCsv/ENC2 for aix2
//     TaskSetupArmControl Inputs/SetupArmControl.m_setupRobot.m_setupArms[4].m_joints[5].m_motorInputs/m_motorEncoder <-> TxPdoMappingCspCsv/Position actual value for aix2
//     TaskSetupArmControl Inputs/SetupArmControl.m_setupRobot.m_setupArms[4].m_joints[5].m_motorInputs/m_statusWord <-> TxPdoMappingCspCsv/Statusword for aix2
//     TaskSetupArmControl Outputs/SetupArmControl.m_setupRobot.m_setupArms[4].m_joints[4].m_motorOutputs/m_cmdCurrent <-> RxPdoMappingCspCsv/Target torque
//     TaskSetupArmControl Outputs/SetupArmControl.m_setupRobot.m_setupArms[4].m_joints[4].m_motorOutputs/m_cmdMotorEncoder <-> RxPdoMappingCspCsv/Target position
//     TaskSetupArmControl Outputs/SetupArmControl.m_setupRobot.m_setupArms[4].m_joints[4].m_motorOutputs/m_controlWord <-> RxPdoMappingCspCsv/Controlword
//     TaskSetupArmControl Outputs/SetupArmControl.m_setupRobot.m_setupArms[4].m_joints[4].m_motorOutputs/m_opMode <-> RxPdoMappingCspCsv/Modes of operation
//     TaskSetupArmControl Outputs/SetupArmControl.m_setupRobot.m_setupArms[4].m_joints[5].m_motorOutputs/m_cmdCurrent <-> RxPdoMappingCspCsv/Target Torque value for aix2
//     TaskSetupArmControl Outputs/SetupArmControl.m_setupRobot.m_setupArms[4].m_joints[5].m_motorOutputs/m_cmdMotorEncoder <-> RxPdoMappingCspCsv/Target position value for aix2
//     TaskSetupArmControl Outputs/SetupArmControl.m_setupRobot.m_setupArms[4].m_joints[5].m_motorOutputs/m_controlWord <-> RxPdoMappingCspCsv/ControlWord for aix2
//   SlaveController/SlaveController Instance <-> SlaveArm4/SlaveJoint1
//     TaskCartControl Inputs/CartControl.m_cartRobot.m_slaveCart.m_carRotaOverhangIO[4] <-> TxPdoMappingCspCsv/digital input
//     TaskSlaveArmControl Inputs/SlaveArmControl.m_slaveRobot.m_slaveArms[4].m_joints[1].m_motorInputs/m_current <-> TxPdoMappingCspCsv/Torque actual value
//     TaskSlaveArmControl Inputs/SlaveArmControl.m_slaveRobot.m_slaveArms[4].m_joints[1].m_motorInputs/m_driverError <-> TxPdoMappingCspCsv/digital input
//     TaskSlaveArmControl Inputs/SlaveArmControl.m_slaveRobot.m_slaveArms[4].m_joints[1].m_motorInputs/m_electriAngleDev <-> TxPdoMappingCspCsv/Velocity actual value
//     TaskSlaveArmControl Inputs/SlaveArmControl.m_slaveRobot.m_slaveArms[4].m_joints[1].m_motorInputs/m_linkEncoder <-> TxPdoMappingCspCsv/ENC2
//     TaskSlaveArmControl Inputs/SlaveArmControl.m_slaveRobot.m_slaveArms[4].m_joints[1].m_motorInputs/m_motorEncoder <-> TxPdoMappingCspCsv/Position actual value
//     TaskSlaveArmControl Inputs/SlaveArmControl.m_slaveRobot.m_slaveArms[4].m_joints[1].m_motorInputs/m_statusWord <-> TxPdoMappingCspCsv/Statusword
//     TaskSlaveArmControl Outputs/SlaveArmControl.m_slaveRobot.m_slaveArms[4].m_joints[1].m_motorOutputs/m_cmdCurrent <-> RxPdoMappingCspCsv/Target torque
//     TaskSlaveArmControl Outputs/SlaveArmControl.m_slaveRobot.m_slaveArms[4].m_joints[1].m_motorOutputs/m_cmdMotorEncoder <-> RxPdoMappingCspCsv/Target position
//     TaskSlaveArmControl Outputs/SlaveArmControl.m_slaveRobot.m_slaveArms[4].m_joints[1].m_motorOutputs/m_controlWord <-> RxPdoMappingCspCsv/Controlword
//     TaskSlaveArmControl Outputs/SlaveArmControl.m_slaveRobot.m_slaveArms[4].m_joints[1].m_motorOutputs/m_opMode <-> RxPdoMappingCspCsv/Modes of operation
//   SlaveController/SlaveController Instance <-> SlaveArm4/SlaveJoint2
//     TaskSetupArmControl Outputs/SetupArmControl.m_setupRobot.m_setupArms[4].m_lightIO <-> RxPdoMappingCspCsv/Target velocity
//     TaskSlaveArmControl Inputs/SlaveArmControl.m_slaveRobot.m_slaveArms[4].m_joints[2].m_motorInputs/m_current <-> TxPdoMappingCspCsv/Torque actual value
//     TaskSlaveArmControl Inputs/SlaveArmControl.m_slaveRobot.m_slaveArms[4].m_joints[2].m_motorInputs/m_driverError <-> TxPdoMappingCspCsv/digital input
//     TaskSlaveArmControl Inputs/SlaveArmControl.m_slaveRobot.m_slaveArms[4].m_joints[2].m_motorInputs/m_electriAngleDev <-> TxPdoMappingCspCsv/Velocity actual value
//     TaskSlaveArmControl Inputs/SlaveArmControl.m_slaveRobot.m_slaveArms[4].m_joints[2].m_motorInputs/m_linkEncoder <-> TxPdoMappingCspCsv/ENC2
//     TaskSlaveArmControl Inputs/SlaveArmControl.m_slaveRobot.m_slaveArms[4].m_joints[2].m_motorInputs/m_motorEncoder <-> TxPdoMappingCspCsv/Position actual value
//     TaskSlaveArmControl Inputs/SlaveArmControl.m_slaveRobot.m_slaveArms[4].m_joints[2].m_motorInputs/m_statusWord <-> TxPdoMappingCspCsv/Statusword
//     TaskSlaveArmControl Outputs/SlaveArmControl.m_slaveRobot.m_slaveArms[4].m_joints[2].m_motorOutputs/m_cmdCurrent <-> RxPdoMappingCspCsv/Target torque
//     TaskSlaveArmControl Outputs/SlaveArmControl.m_slaveRobot.m_slaveArms[4].m_joints[2].m_motorOutputs/m_cmdMotorEncoder <-> RxPdoMappingCspCsv/Target position
//     TaskSlaveArmControl Outputs/SlaveArmControl.m_slaveRobot.m_slaveArms[4].m_joints[2].m_motorOutputs/m_controlWord <-> RxPdoMappingCspCsv/Controlword
//     TaskSlaveArmControl Outputs/SlaveArmControl.m_slaveRobot.m_slaveArms[4].m_joints[2].m_motorOutputs/m_opMode <-> RxPdoMappingCspCsv/Modes of operation
//   SlaveController/SlaveController Instance <-> SlaveArm4/SlaveJoint3
//     TaskCartControl Inputs/CartControl.m_cartRobot.m_slaveCart.m_trocarIO[4] <-> TxPdoMappingCspCsv/digital input
//     TaskSetupArmControl Inputs/SetupArmControl.m_setupRobot.m_setupArms[4].m_adjustIO <-> TxPdoMappingCspCsv/digital input
//     TaskSlaveArmControl Inputs/SlaveArmControl.m_slaveRobot.m_slaveArms[4].m_adjustIO <-> TxPdoMappingCspCsv/digital input
//     TaskSlaveArmControl Inputs/SlaveArmControl.m_slaveRobot.m_slaveArms[4].m_joints[3].m_motorInputs/m_current <-> TxPdoMappingCspCsv/Torque actual value
//     TaskSlaveArmControl Inputs/SlaveArmControl.m_slaveRobot.m_slaveArms[4].m_joints[3].m_motorInputs/m_linkEncoder <-> TxPdoMappingCspCsv/ENC2
//     TaskSlaveArmControl Inputs/SlaveArmControl.m_slaveRobot.m_slaveArms[4].m_joints[3].m_motorInputs/m_motorEncoder <-> TxPdoMappingCspCsv/Position actual value
//     TaskSlaveArmControl Inputs/SlaveArmControl.m_slaveRobot.m_slaveArms[4].m_joints[3].m_motorInputs/m_statusWord <-> TxPdoMappingCspCsv/Statusword
//     TaskSlaveArmControl Outputs/SlaveArmControl.m_slaveRobot.m_slaveArms[4].m_joints[3].m_motorOutputs/m_cmdCurrent <-> RxPdoMappingCspCsv/Target torque
//     TaskSlaveArmControl Outputs/SlaveArmControl.m_slaveRobot.m_slaveArms[4].m_joints[3].m_motorOutputs/m_cmdMotorEncoder <-> RxPdoMappingCspCsv/Target position
//     TaskSlaveArmControl Outputs/SlaveArmControl.m_slaveRobot.m_slaveArms[4].m_joints[3].m_motorOutputs/m_controlWord <-> RxPdoMappingCspCsv/Controlword
//     TaskSlaveArmControl Outputs/SlaveArmControl.m_slaveRobot.m_slaveArms[4].m_joints[3].m_motorOutputs/m_opMode <-> RxPdoMappingCspCsv/Modes of operation
//   SlaveController/SlaveController Instance <-> SlaveArm4/SlaveJoint45
//     TaskSlaveArmControl Inputs/SlaveArmControl.m_slaveRobot.m_slaveArms[4].m_joints[4].m_motorInputs/m_current <-> TxPdoMappingCspCsv/Velocity actual value for aix2
//     TaskSlaveArmControl Inputs/SlaveArmControl.m_slaveRobot.m_slaveArms[4].m_joints[4].m_motorInputs/m_linkEncoder <-> TxPdoMappingCspCsv/ENC2 for aix2
//     TaskSlaveArmControl Inputs/SlaveArmControl.m_slaveRobot.m_slaveArms[4].m_joints[5].m_motorInputs/m_linkEncoder <-> TxPdoMappingCspCsv/ENC2 for aix3
//     TaskSlaveArmControl Inputs/SlaveArmControl.m_slaveRobot.m_slaveArms[4].m_joints[4].m_motorInputs/m_motorEncoder <-> TxPdoMappingCspCsv/Position actual value for aix2
//     TaskSlaveArmControl Inputs/SlaveArmControl.m_slaveRobot.m_slaveArms[4].m_joints[5].m_motorInputs/m_motorEncoder <-> TxPdoMappingCspCsv/Position actual value for aix3
//     TaskSlaveArmControl Inputs/SlaveArmControl.m_slaveRobot.m_slaveArms[4].m_joints[4].m_motorInputs/m_statusWord <-> TxPdoMappingCspCsv/Statusword
//     TaskSlaveArmControl Inputs/SlaveArmControl.m_slaveRobot.m_slaveArms[4].m_joints[5].m_motorInputs/m_statusWord <-> TxPdoMappingCspCsv/Statusword
//     TaskSlaveArmControl Inputs/SlaveArmControl.m_slaveRobot.m_slaveArms[4].m_joints[5].m_motorInputs/m_current <-> TxPdoMappingCspCsv/Torque actual value for aix3
//     TaskSlaveArmControl Inputs/SlaveArmControl.m_slaveRobot.m_slaveArms[4].m_panelInstrumentOnIO <-> TxPdoMappingCspCsv/digital input
//     TaskSlaveArmControl Outputs/SlaveArmControl.m_slaveRobot.m_slaveArms[4].m_joints[4].m_motorOutputs/m_cmdCurrent <-> RxPdoMappingCspCsv/Target Torque value for aix2
//     TaskSlaveArmControl Outputs/SlaveArmControl.m_slaveRobot.m_slaveArms[4].m_joints[5].m_motorOutputs/m_cmdCurrent <-> RxPdoMappingCspCsv/Target Torque value for aix3
//     TaskSlaveArmControl Outputs/SlaveArmControl.m_slaveRobot.m_slaveArms[4].m_joints[4].m_motorOutputs/m_cmdMotorEncoder <-> RxPdoMappingCspCsv/Target position value for aix2
//     TaskSlaveArmControl Outputs/SlaveArmControl.m_slaveRobot.m_slaveArms[4].m_joints[5].m_motorOutputs/m_cmdMotorEncoder <-> RxPdoMappingCspCsv/Target position value for aix3
//     TaskSlaveArmControl Outputs/SlaveArmControl.m_slaveRobot.m_slaveArms[4].m_joints[4].m_motorOutputs/m_controlWord <-> RxPdoMappingCspCsv/Controlword
//     TaskSlaveArmControl Outputs/SlaveArmControl.m_slaveRobot.m_slaveArms[4].m_joints[4].m_motorOutputs/m_opMode <-> RxPdoMappingCspCsv/Modes of operation
//   SlaveController/SlaveController Instance <-> SlaveArm4/SlaveJoint678
//     TaskSlaveArmControl Inputs/SlaveArmControl.m_slaveRobot.m_slaveArms[4].m_joints[6].m_motorInputs/m_current <-> TxPdoMappingCspCsv/Velocity actual value for aix2
//     TaskSlaveArmControl Inputs/SlaveArmControl.m_slaveRobot.m_slaveArms[4].m_joints[6].m_motorInputs/m_linkEncoder <-> TxPdoMappingCspCsv/ENC2 for aix2
//     TaskSlaveArmControl Inputs/SlaveArmControl.m_slaveRobot.m_slaveArms[4].m_joints[7].m_motorInputs/m_linkEncoder <-> TxPdoMappingCspCsv/ENC2 for aix3
//     TaskSlaveArmControl Inputs/SlaveArmControl.m_slaveRobot.m_slaveArms[4].m_joints[8].m_motorInputs/m_linkEncoder <-> TxPdoMappingCspCsv/ENC2 for aix1
//     TaskSlaveArmControl Inputs/SlaveArmControl.m_slaveRobot.m_slaveArms[4].m_joints[6].m_motorInputs/m_motorEncoder <-> TxPdoMappingCspCsv/Position actual value for aix2
//     TaskSlaveArmControl Inputs/SlaveArmControl.m_slaveRobot.m_slaveArms[4].m_joints[7].m_motorInputs/m_motorEncoder <-> TxPdoMappingCspCsv/Position actual value for aix3
//     TaskSlaveArmControl Inputs/SlaveArmControl.m_slaveRobot.m_slaveArms[4].m_joints[6].m_motorInputs/m_statusWord <-> TxPdoMappingCspCsv/Statusword
//     TaskSlaveArmControl Inputs/SlaveArmControl.m_slaveRobot.m_slaveArms[4].m_joints[7].m_motorInputs/m_statusWord <-> TxPdoMappingCspCsv/Statusword
//     TaskSlaveArmControl Inputs/SlaveArmControl.m_slaveRobot.m_slaveArms[4].m_joints[8].m_motorInputs/m_statusWord <-> TxPdoMappingCspCsv/Statusword
//     TaskSlaveArmControl Inputs/SlaveArmControl.m_slaveRobot.m_slaveArms[4].m_joints[7].m_motorInputs/m_current <-> TxPdoMappingCspCsv/Torque actual value for aix3
//     TaskSlaveArmControl Inputs/SlaveArmControl.m_slaveRobot.m_slaveArms[4].m_joints[8].m_motorInputs/m_current <-> TxPdoMappingCspCsv/Torque actual value
//     TaskSlaveArmControl Inputs/SlaveArmControl.m_slaveRobot.m_slaveArms[4].m_joints[8].m_motorInputs/m_motorEncoder <-> TxPdoMappingCspCsv/Position actual value
//     TaskSlaveArmControl Outputs/SlaveArmControl.m_slaveRobot.m_slaveArms[4].m_joints[6].m_motorOutputs/m_cmdCurrent <-> RxPdoMappingCspCsv/Target Torque value for aix2
//     TaskSlaveArmControl Outputs/SlaveArmControl.m_slaveRobot.m_slaveArms[4].m_joints[7].m_motorOutputs/m_cmdCurrent <-> RxPdoMappingCspCsv/Target Torque value for aix3
//     TaskSlaveArmControl Outputs/SlaveArmControl.m_slaveRobot.m_slaveArms[4].m_joints[6].m_motorOutputs/m_cmdMotorEncoder <-> RxPdoMappingCspCsv/Target position value for aix2
//     TaskSlaveArmControl Outputs/SlaveArmControl.m_slaveRobot.m_slaveArms[4].m_joints[7].m_motorOutputs/m_cmdMotorEncoder <-> RxPdoMappingCspCsv/Target position value for aix3
//     TaskSlaveArmControl Outputs/SlaveArmControl.m_slaveRobot.m_slaveArms[4].m_joints[6].m_motorOutputs/m_controlWord <-> RxPdoMappingCspCsv/Controlword
//     TaskSlaveArmControl Outputs/SlaveArmControl.m_slaveRobot.m_slaveArms[4].m_joints[6].m_motorOutputs/m_opMode <-> RxPdoMappingCspCsv/Modes of operation
//     TaskSlaveArmControl Outputs/SlaveArmControl.m_slaveRobot.m_slaveArms[4].m_joints[8].m_motorOutputs/m_cmdCurrent <-> RxPdoMappingCspCsv/Target Torque value
//     TaskSlaveArmControl Outputs/SlaveArmControl.m_slaveRobot.m_slaveArms[4].m_joints[8].m_motorOutputs/m_cmdMotorEncoder <-> RxPdoMappingCspCsv/Target position
//   SlaveController/SlaveController Instance <-> SlaveController/SlaveController Instance
//     TaskCartControl Inputs/CartControl.m_cartDataPool.m_safetyData <-> TaskCartControl Outputs/SafetyCheck.m_safetyCheckData
//     TaskCartControl Inputs/CartControl.m_cartDataPool.m_slaveStatus <-> TaskSlaveArmControl Outputs/SlaveArmControl.m_slaveStatus
//     TaskDynamic Inputs/RobotDynamics.m_instruInfo <-> TaskSlaveArmControl Outputs/SlaveArmControl.m_slaveStatus/m_instruStauts
//     TaskDynamic Inputs/RobotDynamics.m_setupJointData <-> TaskSetupArmControl Outputs/SetupArmControl.m_setupJointsData
//     TaskDynamic Inputs/RobotDynamics.m_slaveJointsData <-> TaskSlaveArmControl Outputs/SlaveArmControl.m_slaveJointsData
//     TaskSafetyCheck Inputs/SafetyCheck.m_cartJointsData <-> TaskCartControl Outputs/CartControl.m_cartJointsData
//     TaskSafetyCheck Inputs/SafetyCheck.m_cartStatus <-> TaskCartControl Outputs/CartControl.m_cartStatus
//     TaskSafetyCheck Inputs/SafetyCheck.m_setupJointsData <-> TaskSetupArmControl Outputs/SetupArmControl.m_setupJointsData
//     TaskSafetyCheck Inputs/SafetyCheck.m_setupStatus <-> TaskSlaveArmControl Outputs/SetupArmControl.m_setupStatus
//     TaskSafetyCheck Inputs/SafetyCheck.m_slaveJointData <-> TaskSlaveArmControl Outputs/SlaveArmControl.m_slaveJointsData
//     TaskSafetyCheck Inputs/SafetyCheck.m_slaveStatus <-> TaskSlaveArmControl Outputs/SlaveArmControl.m_slaveStatus
//     TaskSetupArmControl Inputs/SetupArmControl.m_setupInputDataPool.m_safetyData <-> TaskCartControl Outputs/SafetyCheck.m_safetyCheckData
//     TaskSetupArmControl Inputs/SetupArmControl.m_setupInputDataPool.m_setupJnt3Gravity <-> TaskDynamic Outputs/RobotDynamics.m_setupJnt3Gravity
//     TaskSetupArmControl Inputs/SetupArmControl.m_setupInputDataPool.m_setupJnt5Gravity <-> TaskDynamic Outputs/RobotDynamics.m_setupJnt5Gravity
//     TaskSetupArmControl Inputs/SetupArmControl.m_setupInputDataPool.m_slaveStatus <-> TaskSlaveArmControl Outputs/SlaveArmControl.m_slaveStatus
//     TaskSlaveArmControl Inputs/SlaveArmControl.m_slaveInputDataPool.m_safetyData <-> TaskCartControl Outputs/SafetyCheck.m_safetyCheckData
//     TaskSlaveArmControl Inputs/SlaveArmControl.m_slaveInputDataPool.m_setupStatus <-> TaskSlaveArmControl Outputs/SetupArmControl.m_setupStatus
//     TaskSlaveArmControl Inputs/SlaveArmControl.m_slaveInputDataPool.m_slaveDynaData <-> TaskDynamic Outputs/RobotDynamics.m_slaveDynaData

// ---- DUTs/Enum/E_CartJointState.TcDUT
TYPE E_CartJointState :
(
	CartJointState_Error := 1,
	CartJointState_Init := 2,
	CartJointState_SelfCheck := 3,
	CartJointState_Standby := 4,
	CartJointState_Ready := 5,
	CartJointState_InSurgery := 6,
	CartJointState_SteadyFootDeployment := 7,
	CartJointState_Movement := 8,
	CartJointState_HangAdjust := 9,
	CartJointState_AsepticDeployment := 10,
	CartJointState_RotaOverhang := 11,
	CartJointState_SlowStop := 12,
	CartJointState_StandColuAdjust := 13,
	CartJointState_SupporLeg := 14,
	
	CartJointState_totalNum := CartJointState_SupporLeg
);
END_TYPE

// ---- DUTs/Structure/TasksCommunication/ST_SlaveUIData.TcDUT
// Output from UI controller
// Input to slave arm control task and cart control task  
TYPE ST_SlaveUIData :
STRUCT
	m_slaveArmDisableFlag :ARRAY[1..4] OF BOOL:=[4(FALSE)];
	m_instruUsageWrite :ARRAY[1..4] OF BOOL:=[4(FALSE)];
	m_armInSelfCheck :  ARRAY [1..g_sArmNum] OF BOOL;
	m_armSelfCheckFinshed :  ARRAY [1..g_sArmNum] OF BOOL;
	m_dumpEnergy : UINT:=51;
END_STRUCT
END_TYPE

// ---- DUTs/Enum/E_DriverCtrlWord.TcDUT
TYPE E_DriverCtrlWord :
(
	DriverCtrlWord_INIT := 6,
	DriverCtrlWord_PREOP := 7,
	DriverCtrlWord_OP := 15,
	DriverCtrlWord_FaultReset := 16#8F,
	DriverCtrlWord_halt := 16#10F
);
END_TYPE

// ---- SafetyCheck/ErrRecord/checkDelayTime.TcDUT
TYPE checkDelayTime :
STRUCT
	//motor encoder and joint encoder deviation delay time
	Ti_armJntEncErr:TIME:=T#0.1S;
	//drive error delay time
	Ti_driveErr:TIME:=T#0.1S;
	//joint encoder ununuited delay time
	Ti_linkEncErr:TIME:=T#5S;
	//joint status error delay time 
	Ti_jntStatusErr:TIME:=T#1S;
	//motor current is not update delay time
	Ti_currentIsNotUpdate:TIME:=T#20S;
	//joint postion out of limit
	Ti_outOfLimit:TIME:=T#0.1S;
	//joint follow error delay time
	Ti_armJntFollowErr:TIME:=T#0.1S;
	//joint vel error delay time
	Ti_jntVelErr:TIME:=T#0.05S;
	//joint current error  delay time
	Ti_jntCurrentErr:TIME:=T#3S;
	//fixed point postion change of  master-slave state 
	Ti_fixedPointErr:TIME:=T#0.1S;
	//space pose error  delay time
	Ti_spacePoseErr:TIME:=T#0.1S;
	//commend joint position saltation delay time
	Ti_jntCmdSaltationErr:TIME:=T#0.002S;
	//Deviation between command current and feedback current
	Ti_jntCmdCurrentErr:TIME:=T#0.2S;

	
	Ti_CarDualEncDev:TIME:=T#0.02S;
	Ti_CarDriveErr:TIME:=T#1S;
	Ti_CarActSec:TIME:=T#10S;
	Ti_CarJntStatus:TIME:=T#1S;
	Ti_CarTorMotor:TIME:=T#20S;
	Ti_CaroutofLimit:TIME:=T#0.1S;
	Ti_CarFollowDev:TIME:=T#0.02S;
	Ti_CarJntVel:TIME:=T#0.05S;
	Ti_CarJntCurrent:TIME:=T#1S;
	Ti_CarMZDriveErr:TIME:=T#1S;
END_STRUCT
END_TYPE

// ---- GVLs/CartJoints/GVL_CartControlParameters.TcGVL
{attribute 'global_init_slot' := '49991'} 
{attribute 'qualified_only'}
VAR_GLOBAL
	// filter cut-off frequency for velocity and torque
	g_curJntVelLpfCutoffFreq :LREAL := 30;
	g_cmdJntTrqLpfCutoffFreq :LREAL := 300;
	g_curJntTrqLpfCutoffFreq :LREAL := 300;
	
	g_curBeamStretchJntInitPos :LREAL := 0.972;
	g_maxCartVel :ARRAY [1..4] OF LREAL:= [0.04, 0.05, 0.05, 5*g_deg2Rad];
	
	g_maxJntVel :ARRAY [1..8] OF LREAL:=[0.0025, 0.0025, 2*pi, 2*pi, 0.050, 5*g_deg2Rad, 0.050, 10*g_deg2Rad];
	g_maxJntAcc :ARRAY [1..8] OF LREAL:=[0.0025*2, 0.0025*2, pi*2, pi*2, 0.050*2, 5*g_deg2Rad*1.5, 0.050*1.5, 10*g_deg2Rad*1.5];
	
	g_surgicalOrientPos : ARRAY [1..5, 1..3, 1..4]  OF LREAL := [
		0.1, 0.10, 0.10, 0.10,    0.1, -0.10, 0.10, -0.10,	0.1, 0.10, 0.10, -0.10,
		0.2, 0.20, 0.20, 0.20,    0.2, -0.20, 0.20, -0.20,	0.2, 0.20, 0.20, -0.20,
		0.3, 0.25, 0.30, 0.30,    0.3, -0.25, 0.30, -0.30,	0.3, 0.25, 0.30, -0.30,
		0.4, 0.30, 0.35, 0.35,    0.4, -0.30, 0.35, -0.35,	0.4, 0.30, 0.35, -0.35,
		0.5, 0.35, 0.40, 0.40,    0.5, -0.35, 0.40, -0.40,	0.4, 0.30, 0.35, -0.35];
	
	g_surgicalDrapingPos : ARRAY[1..8] OF LREAL := [0, 0, 0, 0, 0.3, 0, 0.2, 0];
	
	g_jntCtrlAngTolHigh :LREAL :=1*g_deg2Rad;
	
	g_cartInitialHeight : UINT := 1805;
	g_cartOpenHorizonLaserHeight : UINT := 1950;
END_VAR

// ---- GVLs/CartJoints/GVL_CartJointEncoderCaliData.TcGVL
{attribute 'qualified_only'}
// Robot3 --joints parameters of setup arms
VAR_GLOBAL
	// absolute encoder value at minimal joint positon  2873378  289000
	g_minLinkEncoder :ARRAY[1..g_cartJntNum] OF DINT :=[0, 0, 0, 0, 27616627, 78529, 22410851, 114258];
		 
	// absolute encoder value at maximum joint positon
	g_maxLinkEncoder :ARRAY[1..g_cartJntNum] OF DINT :=[0, 0, 0, 0, 24720108, 101778, 24474011, 105483 ];
	
	// absolute encoder value at calibrated positon
	g_caliLinkEncoder :ARRAY[1..g_cartJntNum] OF DINT :=[0, 0, 0, 0, 27616627, 90321, 24474011, 43437];
	
	 // if absolute encoder value cross zeros within joint motion range
	g_linkEncZeroCross :ARRAY[1..g_cartJntNum] OF INT :=[0, 0, 0, 0, 0, 0, 0, 1];
		 

	// abolute encoder expanded limit buffer in case there is calibrtion error at limit position
	g_linkEncLimitBuffer : DINT := 100000;

	// absolute encoder direction
	g_asbEncoderDir :ARRAY[1..g_cartJntNum] OF INT :=[1, 1, 1, 1, -1, 1, -1, -1];
													
	// flag if joint can rotate multiple cycles
	g_multipleCyclesJoint :ARRAY[1..g_cartJntNum] OF INT :=[0, 0, 0, 0, 0, 0, 0, 0];
		 
	// joint position at link encoder calibrated point
	g_linkEncCaliJntPos :ARRAY[1..g_cartJntNum] OF LREAL :=[0.0, 0.0, 0.0, 0.0, 0.0, 0.0, 0, 0.0];
	
	 // joint SDO address
	g_slaveCartNetID: T_AmsNetId:='169.254.45.61.8.1';
	g_slaveCartJointNetPort:ARRAY[1..g_cartJntNum] OF UINT :=[1001,    1002,	1003,	1004,	1005,	1007,	1008,	1009];

END_VAR

// ---- GVLs/CartJoints/GVL_CartMotorParameters.TcGVL
{attribute 'global_init_slot' := '49991'}
{attribute 'qualified_only'}
VAR_GLOBAL CONSTANT
	// encoder resolution
	//TODO: resolution of joint 2/3 need verification
	g_incEncoderRes :ARRAY[1..g_cartJntNum] OF DINT :=[2(65536), 8388608, 8388608, 8388608, 3(65536)];
	g_absEncoderRes :ARRAY[1..g_cartJntNum] OF DINT :=[1, 1, 1, 1, 8192, 131072, 8192,131072];
	
	// reduction ratio
	g_motorReduction :ARRAY[1..g_cartJntNum] OF LREAL :=
		[100.75*2*pi/0.002, 100.75*2*pi/0.002, 40, 40, 
		 2*(2*pi)/0.005, 676.0/49*356, 299.0/14*(2*pi)/0.020, 676.0/49*238];
	g_absEncoderReduction :ARRAY[1..g_cartJntNum] OF LREAL :=[4(1.0), 2*pi/0.002 , 1.0, 2*pi/0.002, 1.0];
	 
	// motor parameters
	g_motorTrqConst :ARRAY[1..g_cartJntNum] OF LREAL :=[ 0.0256, 0.0256, 0.058,0.058,  0.123,0.0292,0.0292,0.0292];
	g_motorMaxCurrent :ARRAY[1..g_cartJntNum] OF LREAL :=[ 41200,41200,50000,50000,  33000,41200,41200,41200];//mA
	
	
	// motor and absEncoder direction
	g_motorDir :ARRAY[1..g_cartJntNum] OF INT :=[1, 1, 1, -1, 1, 1, -1, -1];
																												 
	// joint position limit
	g_minJntPos: vec8d:=[0, 0, 1, 1, 0, -30*g_deg2Rad, 0.002, -160*g_deg2Rad];	
	g_maxJntPos: vec8d:=[0.053, 0.053, 1, 1,  0.69, 30*g_deg2Rad, 0.498, 160*g_deg2Rad];	
	
END_VAR

// ---- GVLs/GVL_InstruCtrlParams.TcGVL
// NOTICE： Use m_instruTypeIdx in FB_Instrument as the array index to get data below
{attribute 'global_init_slot' := '49991'}
VAR_GLOBAL CONSTANT
	
	// instrument types number
	g_instruTypesNum :INT := 14;
	
